IF pressSectionLowerFeltOverrunOperatorSideAlarm THEN
    alarmsDisplay.pressSectionLowerFeltOverrunOperatorSideAlarm := TRUE;
END_IF

IF pressSectionLowerFeltOverrunDriveSideAlarm THEN
    alarmsDisplay.pressSectionLowerFeltOverrunDriveSideAlarm := TRUE;
END_IF


//────────────────────────────────────────────
// PRESS SECTION — GROUP FAULT
//────────────────────────────────────────────
IF pressSectionGroupFaultAlarm THEN
    alarmsDisplay.pressSectionGroupFaultAlarm := TRUE;
END_IF
END_METHOD

METHOD _03_DryingSectionAlarms
VAR_INPUT
END_VAR
(*
    // ─────────────── LUBRIFICATION PUMPS ───────────────
    lubricationPump1FaultAlarm              : BOOL;  // Lubrication pump 1 fault / trip
    lubricationPump2FaultAlarm              : BOOL;  // Lubrication pump 2 fault / trip
    lubricationMinPressureFaultAlarm        : BOOL;  // Minimum pressure not reached / trip
    lubricationMaxPressureFaultAlarm        : BOOL;  // Overpressure in lubrication circuit / trip
	lubricationTankHighTemperatureAlarm 	: BOOL;
	lubricationCircuitHighTemperatureAlarm 	: BOOL;
*)
//==============================================================
// DRYING SECTION — GROUP 1
//==============================================================

//----------------------------
// Drives — Upper (G1)
//----------------------------
IF 	dryingSectionSafetyAlarm THEN
	
	alarmsDisplay.dryingSectionSafetyAlarm := TRUE;
	
END_IF


IF dryingSectionGroup1UpperMasterFaultAlarm THEN
    alarmsDisplay.dryingSectionGroup1UpperMasterFaultAlarm := TRUE;
END_IF

IF dryingSectionGroup1UpperMasterCoolingFaultAlarm THEN
    alarmsDisplay.dryingSectionGroup1UpperMasterCoolingFaultAlarm := TRUE;
END_IF

IF dryingSectionGroup1UpperSlave1FaultAlarm THEN
    alarmsDisplay.dryingSectionGroup1UpperSlave1FaultAlarm := TRUE;
END_IF

IF dryingSectionGroup1UpperSlave1CoolingFaultAlarm THEN
    alarmsDisplay.dryingSectionGroup1UpperSlave1CoolingFaultAlarm := TRUE;
END_IF

IF dryingSectionGroup1UpperSlave2FaultAlarm THEN
    alarmsDisplay.dryingSectionGroup1UpperSlave2FaultAlarm := TRUE;
END_IF

IF dryingSectionGroup1UpperSlave2CoolingFaultAlarm THEN
    alarmsDisplay.dryingSectionGroup1UpperSlave2CoolingFaultAlarm := TRUE;
END_IF

//----------------------------
// Drives — Lower (G1)
//----------------------------
IF dryingSectionGroup1LowerMasterFaultAlarm THEN
    alarmsDisplay.dryingSectionGroup1LowerMasterFaultAlarm := TRUE;
END_IF

IF dryingSectionGroup1LowerMasterCoolingFaultAlarm THEN
    alarmsDisplay.dryingSectionGroup1LowerMasterCoolingFaultAlarm := TRUE;
END_IF

IF dryingSectionGroup1LowerSlave1FaultAlarm THEN
    alarmsDisplay.dryingSectionGroup1LowerSlave1FaultAlarm := TRUE;
END_IF

IF dryingSectionGroup1LowerSlave1CoolingFaultAlarm THEN
    alarmsDisplay.dryingSectionGroup1LowerSlave1CoolingFaultAlarm := TRUE;
END_IF

IF dryingSectionGroup1LowerSlave2FaultAlarm THEN
    alarmsDisplay.dryingSectionGroup1LowerSlave2FaultAlarm := TRUE;
END_IF

IF dryingSectionGroup1LowerSlave2CoolingFaultAlarm THEN
    alarmsDisplay.dryingSectionGroup1LowerSlave2CoolingFaultAlarm := TRUE;
END_IF

//----------------------------
// Fabric overrun protection (G1)
//----------------------------
IF upperDryingSectionGroup1FabricOverrunOperatorSideAlarm THEN
    alarmsDisplay.upperDryingSectionGroup1FabricOverrunOperatorSideAlarm := TRUE;
END_IF

IF upperDryingSectionGroup1FabricOverrunDriveSideAlarm THEN
    alarmsDisplay.upperDryingSectionGroup1FabricOverrunDriveSideAlarm := TRUE;
END_IF

IF lowerDryingSectionGroup1FabricOverrunOperatorSideAlarm THEN
    alarmsDisplay.lowerDryingSectionGroup1FabricOverrunOperatorSideAlarm := TRUE;
END_IF

IF lowerDryingSectionGroup1FabricOverrunDriveSideAlarm THEN
    alarmsDisplay.lowerDryingSectionGroup1FabricOverrunDriveSideAlarm := TRUE;
END_IF

//----------------------------
// Fabric stretcher (G1)
//----------------------------
IF upperDryingSectionGroup1FabricStretcherMotorFaultAlarm THEN
    alarmsDisplay.upperDryingSectionGroup1FabricStretcherMotorFaultAlarm := TRUE;
END_IF

IF lowerDryingSectionGroup1FabricStretcherMotorFaultAlarm THEN
    alarmsDisplay.lowerDryingSectionGroup1FabricStretcherMotorFaultAlarm := TRUE;
END_IF

//----------------------------
// Auxiliaries (G1)
//----------------------------
IF dryingSectionGroup1PickUpRollPosFaultAlarm THEN
    alarmsDisplay.dryingSectionGroup1PickUpRollPosFaultAlarm := TRUE;
END_IF

IF dryingSectionGroup1BabyDryerScraperOscFaultAlarm THEN
    alarmsDisplay.dryingSectionGroup1BabyDryerScraperOscFaultAlarm := TRUE;
END_IF

IF dryingSectionGroup1UpperScraperOscFaultAlarm THEN
    alarmsDisplay.dryingSectionGroup1UpperScraperOscFaultAlarm := TRUE;
END_IF

IF dryingSectionGroup1LowerScraperOscFaultAlarm THEN
    alarmsDisplay.dryingSectionGroup1LowerScraperOscFaultAlarm := TRUE;
END_IF

dryingSectionGroup1PaperBreakAlarm := alarmsDisplay.dryingSectionGroup1PaperBreakAlarm;


//==============================================================
// DRYING SECTION — GROUP 2
//==============================================================

//----------------------------
// Drives — Upper (G2)
//----------------------------
IF dryingSectionGroup2UpperMasterFaultAlarm THEN
    alarmsDisplay.dryingSectionGroup2UpperMasterFaultAlarm := TRUE;
END_IF

IF dryingSectionGroup2UpperMasterCoolingFaultAlarm THEN
    alarmsDisplay.dryingSectionGroup2UpperMasterCoolingFaultAlarm := TRUE;
END_IF

IF dryingSectionGroup2UpperSlave1FaultAlarm THEN
    alarmsDisplay.dryingSectionGroup2UpperSlave1FaultAlarm := TRUE;
END_IF

IF dryingSectionGroup2UpperSlave1CoolingFaultAlarm THEN
    alarmsDisplay.dryingSectionGroup2UpperSlave1CoolingFaultAlarm := TRUE;
END_IF

IF dryingSectionGroup2UpperSlave2FaultAlarm THEN
    alarmsDisplay.dryingSectionGroup2UpperSlave2FaultAlarm := TRUE;
END_IF

IF dryingSectionGroup2UpperSlave2CoolingFaultAlarm THEN
    alarmsDisplay.dryingSectionGroup2UpperSlave2CoolingFaultAlarm := TRUE;
END_IF

//----------------------------
// Drives — Lower (G2)
//----------------------------
IF dryingSectionGroup2LowerMasterFaultAlarm THEN
    alarmsDisplay.dryingSectionGroup2LowerMasterFaultAlarm := TRUE;
END_IF

IF dryingSectionGroup2LowerMasterCoolingFaultAlarm THEN
    alarmsDisplay.dryingSectionGroup2LowerMasterCoolingFaultAlarm := TRUE;
END_IF

IF dryingSectionGroup2LowerSlave1FaultAlarm THEN
    alarmsDisplay.dryingSectionGroup2LowerSlave1FaultAlarm := TRUE;
END_IF

IF dryingSectionGroup2LowerSlave1CoolingFaultAlarm THEN
    alarmsDisplay.dryingSectionGroup2LowerSlave1CoolingFaultAlarm := TRUE;
END_IF

IF dryingSectionGroup2LowerSlave2FaultAlarm THEN
    alarmsDisplay.dryingSectionGroup2LowerSlave2FaultAlarm := TRUE;
END_IF

IF dryingSectionGroup2LowerSlave2CoolingFaultAlarm THEN
    alarmsDisplay.dryingSectionGroup2LowerSlave2CoolingFaultAlarm := TRUE;
END_IF

//----------------------------
// Fabric overrun protection (G2)
//----------------------------
IF upperDryingSectionGroup2FabricOverrunOperatorSideAlarm THEN
    alarmsDisplay.upperDryingSectionGroup2FabricOverrunOperatorSideAlarm := TRUE;
END_IF

IF upperDryingSectionGroup2FabricOverrunDriveSideAlarm THEN
    alarmsDisplay.upperDryingSectionGroup2FabricOverrunDriveSideAlarm := TRUE;
END_IF

IF lowerDryingSectionGroup2FabricOverrunOperatorSideAlarm THEN
    alarmsDisplay.lowerDryingSectionGroup2FabricOverrunOperatorSideAlarm := TRUE;
END_IF

IF lowerDryingSectionGroup2FabricOverrunDriveSideAlarm THEN
    alarmsDisplay.lowerDryingSectionGroup2FabricOverrunDriveSideAlarm := TRUE;
END_IF

//----------------------------
// Fabric stretcher (G2)
//----------------------------
IF upperDryingSectionGroup2FabricStretcherMotorFaultAlarm THEN
    alarmsDisplay.upperDryingSectionGroup2FabricStretcherMotorFaultAlarm := TRUE;
END_IF

IF lowerDryingSectionGroup2FabricStretcherMotorFaultAlarm THEN
    alarmsDisplay.lowerDryingSectionGroup2FabricStretcherMotorFaultAlarm := TRUE;
END_IF

//----------------------------
// Auxiliaries (G2)
//----------------------------
IF dryingSectionGroup2PickUpRollPosFaultAlarm THEN
    alarmsDisplay.dryingSectionGroup2PickUpRollPosFaultAlarm := TRUE;
END_IF

IF dryingSectionGroup2BabyDryerScraperOscFaultAlarm THEN
    alarmsDisplay.dryingSectionGroup2BabyDryerScraperOscFaultAlarm := TRUE;
END_IF

IF dryingSectionGroup2UpperScraperOscFaultAlarm THEN
    alarmsDisplay.dryingSectionGroup2UpperScraperOscFaultAlarm := TRUE;
END_IF

IF dryingSectionGroup2LowerScraperOscFaultAlarm THEN
    alarmsDisplay.dryingSectionGroup2LowerScraperOscFaultAlarm := TRUE;
END_IF

IF dryingSectionGroup2PaperBreakAlarm THEN
    alarmsDisplay.dryingSectionGroup2PaperBreakAlarm := TRUE;
END_IF


//==============================================================
// DRYING SECTION — GROUP 3
//==============================================================

//----------------------------
// Drives — Upper (G3)
//----------------------------
IF dryingSectionGroup3UpperMasterFaultAlarm THEN
    alarmsDisplay.dryingSectionGroup3UpperMasterFaultAlarm := TRUE;
END_IF

IF dryingSectionGroup3UpperMasterCoolingFaultAlarm THEN
    alarmsDisplay.dryingSectionGroup3UpperMasterCoolingFaultAlarm := TRUE;
END_IF

IF dryingSectionGroup3UpperSlave1FaultAlarm THEN
    alarmsDisplay.dryingSectionGroup3UpperSlave1FaultAlarm := TRUE;
END_IF

IF dryingSectionGroup3UpperSlave1CoolingFaultAlarm THEN
    alarmsDisplay.dryingSectionGroup3UpperSlave1CoolingFaultAlarm := TRUE;
END_IF

IF dryingSectionGroup3UpperSlave2FaultAlarm THEN
    alarmsDisplay.dryingSectionGroup3UpperSlave2FaultAlarm := TRUE;
END_IF

IF dryingSectionGroup3UpperSlave2CoolingFaultAlarm THEN
    alarmsDisplay.dryingSectionGroup3UpperSlave2CoolingFaultAlarm := TRUE;
END_IF

//----------------------------
// Drives — Lower (G3)
//----------------------------
IF dryingSectionGroup3LowerMasterFaultAlarm THEN
    alarmsDisplay.dryingSectionGroup3LowerMasterFaultAlarm := TRUE;
END_IF

IF dryingSectionGroup3LowerMasterCoolingFaultAlarm THEN
    alarmsDisplay.dryingSectionGroup3LowerMasterCoolingFaultAlarm := TRUE;
END_IF

IF dryingSectionGroup3LowerSlave1FaultAlarm THEN
    alarmsDisplay.dryingSectionGroup3LowerSlave1FaultAlarm := TRUE;
END_IF

IF dryingSectionGroup3LowerSlave1CoolingFaultAlarm THEN
    alarmsDisplay.dryingSectionGroup3LowerSlave1CoolingFaultAlarm := TRUE;
END_IF

IF dryingSectionGroup3LowerSlave2FaultAlarm THEN
    alarmsDisplay.dryingSectionGroup3LowerSlave2FaultAlarm := TRUE;
END_IF

IF dryingSectionGroup3LowerSlave2CoolingFaultAlarm THEN
    alarmsDisplay.dryingSectionGroup3LowerSlave2CoolingFaultAlarm := TRUE;
END_IF

//----------------------------
// Fabric overrun protection (G3)
//----------------------------
IF upperDryingSectionGroup3FabricOverrunOperatorSideAlarm THEN
    alarmsDisplay.upperDryingSectionGroup3FabricOverrunOperatorSideAlarm := TRUE;
END_IF

IF upperDryingSectionGroup3FabricOverrunDriveSideAlarm THEN
    alarmsDisplay.upperDryingSectionGroup3FabricOverrunDriveSideAlarm := TRUE;
END_IF

IF lowerDryingSectionGroup3FabricOverrunOperatorSideAlarm THEN
    alarmsDisplay.lowerDryingSectionGroup3FabricOverrunOperatorSideAlarm := TRUE;
END_IF

IF lowerDryingSectionGroup3FabricOverrunDriveSideAlarm THEN
    alarmsDisplay.lowerDryingSectionGroup3FabricOverrunDriveSideAlarm := TRUE;
END_IF

//----------------------------
// Fabric stretcher (G3)
//----------------------------
IF upperDryingSectionGroup3FabricStretcherMotorFaultAlarm THEN
    alarmsDisplay.upperDryingSectionGroup3FabricStretcherMotorFaultAlarm := TRUE;
END_IF

IF lowerDryingSectionGroup3FabricStretcherMotorFaultAlarm THEN
    alarmsDisplay.lowerDryingSectionGroup3FabricStretcherMotorFaultAlarm := TRUE;
END_IF

//----------------------------
// Auxiliaries (G3)
//----------------------------
IF dryingSectionGroup3PickUpRollPosFaultAlarm THEN
    alarmsDisplay.dryingSectionGroup3PickUpRollPosFaultAlarm := TRUE;
END_IF

IF dryingSectionGroup3BabyDryerScraperOscFaultAlarm THEN
    alarmsDisplay.dryingSectionGroup3BabyDryerScraperOscFaultAlarm := TRUE;
END_IF

IF dryingSectionGroup3UpperScraperOscFaultAlarm THEN
    alarmsDisplay.dryingSectionGroup3UpperScraperOscFaultAlarm := TRUE;
END_IF

IF dryingSectionGroup3LowerScraperOscFaultAlarm THEN
    alarmsDisplay.dryingSectionGroup3LowerScraperOscFaultAlarm := TRUE;
END_IF

IF dryingSectionGroup3PaperBreakAlarm THEN
    alarmsDisplay.dryingSectionGroup3PaperBreakAlarm := TRUE;
END_IF

IF lubricationMinPressureFaultAlarm THEN
	
	alarmsDisplay.lubricationMinPressureFaultAlarm := TRUE;
	
END_IF

IF lubricationMaxPressureFaultAlarm THEN
	
	alarmsDisplay.lubricationMaxPressureFaultAlarm := TRUE;
	
END_IF



IF lubricationPump1FaultAlarm THEN
	
	alarmsDisplay.lubricationPump1FaultAlarm := TRUE;
	
END_IF

IF lubricationPump2FaultAlarm THEN
	
	alarmsDisplay.lubricationPump2FaultAlarm := TRUE;
	
END_IF

IF lubricationTankHighTemperatureAlarm THEN
	
	alarmsDisplay.lubricationTankHighTemperatureAlarm := TRUE;
	
END_IF


IF lubricationCircuitHighTemperatureAlarm THEN
	
	alarmsDisplay.lubricationCircuitHighTemperatureAlarm := TRUE;
	
END_IF
END_METHOD

METHOD _04_WinderSectionAlarms
VAR_INPUT
END_VAR
(*

    // ─────────────── DRYING SECTION — GROUP 1 ───────────────
    dryingSectionGroup1UpperMasterFaultAlarm         : BOOL;  // G1 Upper Master fault / trip
    dryingSectionGroup1UpperMasterCoolingFaultAlarm  : BOOL;  // G1 Upper Master forced cooling fault
    dryingSectionGroup1UpperSlave1FaultAlarm         : BOOL;  // G1 Upper Slave1 fault / trip
    dryingSectionGroup1UpperSlave1CoolingFaultAlarm  : BOOL;  // G1 Upper Slave1 forced cooling fault
    dryingSectionGroup1UpperSlave2FaultAlarm         : BOOL;  // G1 Upper Slave2 fault / trip
    dryingSectionGroup1UpperSlave2CoolingFaultAlarm  : BOOL;  // G1 Upper Slave2 forced cooling fault

    dryingSectionGroup1LowerMasterFaultAlarm         : BOOL;  // G1 Lower Master fault / trip
    dryingSectionGroup1LowerMasterCoolingFaultAlarm  : BOOL;  // G1 Lower Master forced cooling fault
    dryingSectionGroup1LowerSlave1FaultAlarm         : BOOL;  // G1 Lower Slave1 fault / trip
    dryingSectionGroup1LowerSlave1CoolingFaultAlarm  : BOOL;  // G1 Lower Slave1 forced cooling fault
    dryingSectionGroup1LowerSlave2FaultAlarm         : BOOL;  // G1 Lower Slave2 fault / trip
    dryingSectionGroup1LowerSlave2CoolingFaultAlarm  : BOOL;  // G1 Lower Slave2 forced cooling fault

    // ── FABRIC OVERRUN PROTECTION — GROUP 1 ───────────────────────────────────
    upperDryingSectionGroup1FabricOverrunOperatorSideAlarm : BOOL;  // Fabric overrun detected on operator side (sensor active)
    upperDryingSectionGroup1FabricOverrunDriveSideAlarm    : BOOL;  // Fabric overrun detected on drive side (sensor active)
    lowerDryingSectionGroup1FabricOverrunOperatorSideAlarm : BOOL;  // Fabric overrun detected on operator side (sensor active)
    lowerDryingSectionGroup1FabricOverrunDriveSideAlarm    : BOOL;  // Fabric overrun detected on drive side (sensor active)

    // ───────── DRYING SECTION — FABRIC STRETCHER — GROUP 1 ─────────
    upperDryingSectionGroup1FabricStretcherMotorFaultAlarm : BOOL;  // Upper fabric stretcher motor fault (G1)
    lowerDryingSectionGroup1FabricStretcherMotorFaultAlarm : BOOL;  // Lower fabric stretcher motor fault (G1)

    // ───────── DRYING SECTION — AUXILIARIES — GROUP 1 ─────────
    dryingSectionGroup1PickUpRollPosFaultAlarm       : BOOL;  // EN: G1 pick-up roll positioner fault / PT: Falha do posicionador do rolo pick-up G1
    dryingSectionGroup1BabyDryerScraperOscFaultAlarm : BOOL;  // EN: G1 babydryer scraper oscillator fault / PT: Falha do oscilador da raspa do babydryer G1
    dryingSectionGroup1UpperScraperOscFaultAlarm     : BOOL;  // EN: G1 upper group scraper oscillator fault / PT: Falha do oscilador da raspa do grupo superior G1
    dryingSectionGroup1LowerScraperOscFaultAlarm     : BOOL;  // EN: G1 lower group scraper oscillator fault / PT: Falha do oscilador da raspa do grupo inferior G1
    dryingSectionGroup1PaperBreakAlarm     : BOOL;  // EN: G1 lower group scraper oscillator fault / PT: Falha do oscilador da raspa do grupo inferior G1

    // ─────────────── DRYING SECTION — GROUP 2 ───────────────
    dryingSectionGroup2UpperMasterFaultAlarm         : BOOL;  // G2 Upper Master fault / trip
    dryingSectionGroup2UpperMasterCoolingFaultAlarm  : BOOL;  // G2 Upper Master forced cooling fault
    dryingSectionGroup2UpperSlave1FaultAlarm         : BOOL;  // G2 Upper Slave1 fault / trip
    dryingSectionGroup2UpperSlave1CoolingFaultAlarm  : BOOL;  // G2 Upper Slave1 forced cooling fault
    dryingSectionGroup2UpperSlave2FaultAlarm         : BOOL;  // G2 Upper Slave2 fault / trip
    dryingSectionGroup2UpperSlave2CoolingFaultAlarm  : BOOL;  // G2 Upper Slave2 forced cooling fault

    dryingSectionGroup2LowerMasterFaultAlarm         : BOOL;  // G2 Lower Master fault / trip
    dryingSectionGroup2LowerMasterCoolingFaultAlarm  : BOOL;  // G2 Lower Master forced cooling fault
    dryingSectionGroup2LowerSlave1FaultAlarm         : BOOL;  // G2 Lower Slave1 fault / trip
    dryingSectionGroup2LowerSlave1CoolingFaultAlarm  : BOOL;  // G2 Lower Slave1 forced cooling fault
    dryingSectionGroup2LowerSlave2FaultAlarm         : BOOL;  // G2 Lower Slave2 fault / trip
    dryingSectionGroup2LowerSlave2CoolingFaultAlarm  : BOOL;  // G2 Lower Slave2 forced cooling fault

    // ── FABRIC OVERRUN PROTECTION — GROUP 2 ───────────────────────────────────
    upperDryingSectionGroup2FabricOverrunOperatorSideAlarm : BOOL;  // Fabric overrun detected on operator side (sensor active)
    upperDryingSectionGroup2FabricOverrunDriveSideAlarm    : BOOL;  // Fabric overrun detected on drive side (sensor active)
    lowerDryingSectionGroup2FabricOverrunOperatorSideAlarm : BOOL;  // Fabric overrun detected on operator side (sensor active)
    lowerDryingSectionGroup2FabricOverrunDriveSideAlarm    : BOOL;  // Fabric overrun detected on drive side (sensor active)

    // ───────── DRYING SECTION — FABRIC STRETCHER — GROUP 2 ─────────
    upperDryingSectionGroup2FabricStretcherMotorFaultAlarm : BOOL;  // Upper fabric stretcher motor fault (G2)
    lowerDryingSectionGroup2FabricStretcherMotorFaultAlarm : BOOL;  // Lower fabric stretcher motor fault (G2)

    // ───────── DRYING SECTION — AUXILIARIES — GROUP 2 ─────────
    dryingSectionGroup2PickUpRollPosFaultAlarm       : BOOL;  // EN: G2 pick-up roll positioner fault / PT: Falha do posicionador do rolo pick-up G2
    dryingSectionGroup2BabyDryerScraperOscFaultAlarm : BOOL;  // EN: G2 babydryer scraper oscillator fault / PT: Falha do oscilador da raspa do babydryer G2
    dryingSectionGroup2UpperScraperOscFaultAlarm     : BOOL;  // EN: G2 upper group scraper oscillator fault / PT: Falha do oscilador da raspa do grupo superior G2
    dryingSectionGroup2LowerScraperOscFaultAlarm     : BOOL;  // EN: G2 lower group scraper oscillator fault / PT: Falha do oscilador da raspa do grupo inferior G2
    dryingSectionGroup2PaperBreakAlarm     : BOOL;  // EN: G1 lower group scraper oscillator fault / PT: Falha do oscilador da raspa do grupo inferior G1

    // ─────────────── DRYING SECTION — GROUP 3 ───────────────
    dryingSectionGroup3UpperMasterFaultAlarm         : BOOL;  // G3 Upper Master fault / trip
    dryingSectionGroup3UpperMasterCoolingFaultAlarm  : BOOL;  // G3 Upper Master forced cooling fault
    dryingSectionGroup3UpperSlave1FaultAlarm         : BOOL;  // G3 Upper Slave1 fault / trip
    dryingSectionGroup3UpperSlave1CoolingFaultAlarm  : BOOL;  // G3 Upper Slave1 forced cooling fault
    dryingSectionGroup3UpperSlave2FaultAlarm         : BOOL;  // G3 Upper Slave2 fault / trip
    dryingSectionGroup3UpperSlave2CoolingFaultAlarm  : BOOL;  // G3 Upper Slave2 forced cooling fault

    dryingSectionGroup3LowerMasterFaultAlarm         : BOOL;  // G3 Lower Master fault / trip
    dryingSectionGroup3LowerMasterCoolingFaultAlarm  : BOOL;  // G3 Lower Master forced cooling fault
    dryingSectionGroup3LowerSlave1FaultAlarm         : BOOL;  // G3 Lower Slave1 fault / trip
    dryingSectionGroup3LowerSlave1CoolingFaultAlarm  : BOOL;  // G3 Lower Slave1 forced cooling fault
    dryingSectionGroup3LowerSlave2FaultAlarm         : BOOL;  // G3 Lower Slave2 fault / trip
    dryingSectionGroup3LowerSlave2CoolingFaultAlarm  : BOOL;  // G3 Lower Slave2 forced cooling fault

    // ── FABRIC OVERRUN PROTECTION — GROUP 3 ───────────────────────────────────
    upperDryingSectionGroup3FabricOverrunOperatorSideAlarm : BOOL;  // Fabric overrun detected on operator side (sensor active)
    upperDryingSectionGroup3FabricOverrunDriveSideAlarm    : BOOL;  // Fabric overrun detected on drive side (sensor active)
    lowerDryingSectionGroup3FabricOverrunOperatorSideAlarm : BOOL;  // Fabric overrun detected on operator side (sensor active)
    lowerDryingSectionGroup3FabricOverrunDriveSideAlarm    : BOOL;  // Fabric overrun detected on drive side (sensor active)

    // ───────── DRYING SECTION — FABRIC STRETCHER — GROUP 3 ─────────
    upperDryingSectionGroup3FabricStretcherMotorFaultAlarm : BOOL;  // Upper fabric stretcher motor fault (G3)
    lowerDryingSectionGroup3FabricStretcherMotorFaultAlarm : BOOL;  // Lower fabric stretcher motor fault (G3)

    // ───────── DRYING SECTION — AUXILIARIES — GROUP 3 ─────────
    dryingSectionGroup3PickUpRollPosFaultAlarm       : BOOL;  // EN: G3 pick-up roll positioner fault / PT: Falha do posicionador do rolo pick-up G3
    dryingSectionGroup3BabyDryerScraperOscFaultAlarm : BOOL;  // EN: G3 babydryer scraper oscillator fault / PT: Falha do oscilador da raspa do babydryer G3
    dryingSectionGroup3UpperScraperOscFaultAlarm     : BOOL;  // EN: G3 upper group scraper oscillator fault / PT: Falha do oscilador da raspa do grupo superior G3
    dryingSectionGroup3LowerScraperOscFaultAlarm     : BOOL;  // EN: G3 lower group scraper oscillator fault / PT: Falha do oscilador da raspa do grupo inferior G3
    dryingSectionGroup3PaperBreakAlarm     : BOOL;  // EN: G1 lower group scraper oscillator fault / PT: Falha do oscilador da raspa do grupo inferior G1

*)
//==============================================================
// DRYING SECTION — GROUP 1
//==============================================================

//----------------------------
// Drives — Upper (G1)
//----------------------------
IF 	winderSectionSafetyAlarm THEN
	
	alarmsDisplay.winderSectionSafetyAlarm := TRUE;
	
END_IF
END_METHOD

METHOD _08_AlarmIndication

VAR
	
	alarmCompResult	: DINT;

END_VAR

alarmCompResult := MEMCMP(pBuf1:= ADR(alarmsVariables) , pBuf2:= ADR(alarmsDisplay) , n:= SIZEOF(alarmsDisplay));

//alarmCompResult := alarmsVariables <> alarmsDisplay;

IF alarmCompResult <> 0 THEN

	alarmIndication := TRUE;
ELSE
	
	alarmIndication := FALSE;
	
END_IF
END_METHOD

END_FUNCTION_BLOCK

// ---- Function Blocks/DELTA - MS300/FB_DELTA_C2000_ETC.TcPOU
FUNCTION_BLOCK FB_DELTA_C2000_ETC



//======================================================================
// Persistent Configuration Inputs
//======================================================================
VAR_INPUT PERSISTENT
	
    deviceConfig            : C2000_DEV_CONFIG;       // Device-specific configuration (scaling, limits, etc.)

END_VAR

//======================================================================
// Runtime Inputs
//======================================================================
VAR_INPUT
	
    speedSetpoint           : REAL;                		// Motor speed reference to be written to drive
	torqueSetpoint			: REAL;						// Torque limit if running as torque
    commandWord             : C2000_CONTROLWORD;      	// Control word to drive (start, stop, etc.)
    digitalOutputs          : C2000_DIGITAL_OUTPUTS;  	// Digital output values to send to drive
    analogOutputs           : C2000_ANALOG_OUTPUTS;   	// Analog output values to send to drive
	
END_VAR

//======================================================================
// Runtime Outputs
//======================================================================
VAR_OUTPUT
	
    statusWord              : C2000_STATUSWORD;       // Current status word read from drive
    digitalInputs           : C2000_DIGITAL_INPUTS;   // Current status of digital inputs from drive
    analogInputs            : C2000_ANALOG_INPUTS;    // Current status of analog inputs from drive
    motorSpeedRPM             : REAL;                   // Actual motor speed read from drive in RPM
    motorSpeedEng             : REAL;                   // Actual motor speed read from drive in enginering units scaled
    outputCurrent           : REAL;                   // Output current read from drive
    outputTorque            : REAL;                   // Output torque read from drive
	
	
	pdoSpeedSet			: INT;
	
	
END_VAR

//======================================================================
// Internal Variables
//======================================================================
VAR
    PDOS                    : C2000_PDOS;             // Process Data Object structure containing drive mappings
    // One-shot + pulse for fault reset
    rTrigReset : R_TRIG;
    tReset     : TOF;
	
    // Base OMS bits default (keep your logic)
    b0_swOn, b1_enVolt, b2_qStopOK, b3_enOp : BOOL;
    b4, b5, b6, b7_faultReset, b8_halt      : BOOL;
    cw                                       : WORD;

    // Reset sequencer helpers
 //   rTrigReset        : R_TRIG;   // detect rising edge of reset command
    tResetClear       : TON;      // phase 1: clear all bits (control word = 0)
    tResetPulse       : TON;      // phase 2: pulse bit7 = 1
    resetSeqActive    : BOOL;     // TRUE while running either phase
    resetClearPt      : TIME := T#500MS;    // adjust if your drive needs longer clear
    resetPulsePt      : TIME := T#1000ms;  // 1 second fault-reset pulse	

END_VAR

(*==============================================================================================================================
CPNTeck - Automação Industrial
(c)Copyright 2025 All Rights Reserved
_______________________________________________________________________________________________________________________________
Library: N/A
Tested with: CX920
Engineering: TwinCAT 3
Restrictions: -
Requirements: N/A
Functionality: This function block communicates with a Delta MS300 drive over Modbus RTU. It reads process values such as
               motor speed, current, torque, status words, digital and analog inputs, and writes control commands and 
               setpoints to the drive. The block includes timeout monitoring and state-based communication handling.
Support: fabio@cpnteck.com.br
Note: Parameter comments are only available in language 'English (United States)'

_______________________________________________________________________________________________________________________________
Change log table:

Version         | Date         | Expert in charge   | Changes applied
01.00.01        | 31.05.2025   | Fabio Campion      | Initial implementation for MS300 drive Modbus RTU communication
==============================================================================================================================*)

_StatusWord();       // Method to handle the status word of the drive
_DigitalInputs();    // Method to process the status of digital inputs
_AnalogInputs();     // Method to handle analog input values

_CommandWord();      // Method to set or process the command word for the drive
_DigitalOutputs();   // Method to manage the status of digital outputs
_AnalogOutputs();    // Method to handle analog output values
_SetOperationMode();
_FeedBackVariables(); // Method to process feedback variables from the drive
_SpeedReference();         // Method to set or process the setpoint values
_TorqueReference();

METHOD PRIVATE _AnalogInputs
VAR_INPUT
END_VAR
END_METHOD

METHOD PRIVATE _AnalogOutputs
VAR_INPUT
END_VAR
END_METHOD

METHOD PRIVATE _CommandWord
VAR_INPUT
END_VAR
(*
VAR
    // Internal
    b0_swOn, b1_enVolt, b2_qStopOK, b3_enOp, b4, b5, b6 : BOOL;
    b7_faultReset, b8_halt                              : BOOL;
    cw                                                  : UINT;
END_VAR
*)

b4 := 1;
b5 := 1;
b6 := 1;


// ---------- 1) Base state from commands (bits 0..3) ----------
IF commandWord.quickStop THEN
    // Quick-stop has highest priority: keep voltage/switch-on, clear enable op, force bit2=0
    b0_swOn    := TRUE;
    b1_enVolt  := TRUE;
    b2_qStopOK := FALSE;  // bit2=0 => quick stop active
    b3_enOp    := FALSE;

ELSIF commandWord.enableDrive THEN
    // Enable Operation: 1,1,1,1
    b0_swOn    := TRUE;
    b1_enVolt  := TRUE;
    b2_qStopOK := TRUE;
    b3_enOp    := TRUE;

ELSIF commandWord.stopRequest THEN
    // Switch On (ready but not enabled): 1,1,1,0
    b0_swOn    := TRUE;
    b1_enVolt  := TRUE;
    b2_qStopOK := TRUE;
    b3_enOp    := FALSE;

ELSE
    // Shutdown (safe, DC bus on): 0,1,1,0
    b0_swOn    := FALSE;
    b1_enVolt  := TRUE;
    b2_qStopOK := TRUE;
    b3_enOp    := FALSE;
END_IF


// ---------- 2) Halt (bit8) ----------
b8_halt := commandWord.halt;

// ---------- 3) Fault Reset as 1000 ms pulse (bit7) ----------
rTrigReset(CLK := commandWord.faultResetCmd);
tReset(IN := rTrigReset.Q, PT := T#1000ms);
b7_faultReset := tReset.Q;

// ---------- 4) Pack bits into 16-bit control word ----------
cw := 0; // bits 9..15 remain 0 unless you set them later

// base (0..3)
IF b0_swOn    THEN cw := cw OR 16#0001; END_IF; // bit0
IF b1_enVolt  THEN cw := cw OR 16#0002; END_IF; // bit1
IF b2_qStopOK THEN cw := cw OR 16#0004; END_IF; // bit2
IF b3_enOp    THEN cw := cw OR 16#0008; END_IF; // bit3

// OMS (4..6) — use correct masks
IF b4          THEN cw := cw OR 16#0010; END_IF; // bit4
IF b5          THEN cw := cw OR 16#0020; END_IF; // bit5
IF b6          THEN cw := cw OR 16#0040; END_IF; // bit6

// bit7 (fault reset pulse) and bit8 (halt)
IF b7_faultReset THEN cw := cw OR 16#0080; END_IF; // bit7
IF b8_halt       THEN cw := cw OR 16#0100; END_IF; // bit8

// Bits 9..15 reserved = 0
PDOS.PlcToDrv.controlWord := cw;



//==============================================================
// CIA402 CONTROL WORD BUILD — with proper reset sequence
//==============================================================
(*

//==============================================================
// 0) Edge-detect RESET command and run the two-phase sequence
//==============================================================
rTrigReset(CLK := commandWord.faultResetCmd);

// Start sequence on rising edge
IF rTrigReset.Q THEN
    resetSeqActive := TRUE;
    // (Re)start clear phase
    tResetClear(IN := TRUE, PT := resetClearPt);
    // ensure pulse is off until clear finishes
    tResetPulse(IN := FALSE, PT := resetPulsePt);
END_IF;

// Advance/reset timers when sequence is active
IF resetSeqActive THEN
    // Phase 1: CLEAR (control word = 0)
    tResetClear(IN := tResetClear.IN, PT := resetClearPt);

    // When clear finishes, start pulse (only once)
    IF tResetClear.Q AND NOT tResetPulse.IN THEN
        tResetClear(IN := FALSE, PT := resetClearPt);     // stop clear timer
        tResetPulse(IN := TRUE,  PT := resetPulsePt);     // start pulse
    END_IF;

    // Run pulse
    tResetPulse(IN := tResetPulse.IN, PT := resetPulsePt);

    // Sequence ends when pulse finishes
    IF tResetPulse.Q THEN
        tResetPulse(IN := FALSE, PT := resetPulsePt);
        resetSeqActive := FALSE;
    END_IF;
END_IF;


//==============================================================
// 1) NORMAL PACKING (only used when NOT resetting)
//==============================================================

// Default OMS high (per your original)
b4 := TRUE;  // bit4 mask 0x0010
b5 := TRUE;  // bit5 mask 0x0020
b6 := TRUE;  // bit6 mask 0x0040

// ---------- 1) Base state from commands (bits 0..3) ----------
IF commandWord.quickStop THEN
    // Quick-stop has highest priority
    b0_swOn    := TRUE;
    b1_enVolt  := TRUE;
    b2_qStopOK := FALSE; // quick stop active
    b3_enOp    := FALSE;

ELSIF commandWord.enableDrive THEN
    // Enable Operation: 1,1,1,1
    b0_swOn    := TRUE;
    b1_enVolt  := TRUE;
    b2_qStopOK := TRUE;
    b3_enOp    := TRUE;

ELSIF commandWord.stopRequest THEN
    // Switch On (ready but not enabled): 1,1,1,0
    b0_swOn    := TRUE;
    b1_enVolt  := TRUE;
    b2_qStopOK := TRUE;
    b3_enOp    := FALSE;

ELSE
    // Shutdown (safe, DC bus on): 0,1,1,0
    b0_swOn    := FALSE;
    b1_enVolt  := TRUE;
    b2_qStopOK := TRUE;
    b3_enOp    := FALSE;
END_IF;

// ---------- 2) Halt (bit8) ----------
b8_halt := commandWord.halt;


//==============================================================
// 2) BUILD CONTROL WORD — with RESET SEQUENCE OVERRIDE
//==============================================================
cw := 0;

// If reset sequence is active, override everything
IF resetSeqActive THEN
    // Phase 1: CLEAR → send 0x0000
    IF NOT tResetClear.Q THEN
//        cw := 16#0000;
        cw := 16#0080;
		

    // Phase 2: PULSE → send only bit7 = 1 (0x0080)
    ELSIF tResetClear.Q AND NOT tResetPulse.Q THEN
//        cw := 16#0080;
        cw := 16#0000;
		
    END_IF;

ELSE
    // Normal packing
    // base (0..3)
    IF b0_swOn    THEN cw := cw OR 16#0001; END_IF; // bit0
    IF b1_enVolt  THEN cw := cw OR 16#0002; END_IF; // bit1
    IF b2_qStopOK THEN cw := cw OR 16#0004; END_IF; // bit2
    IF b3_enOp    THEN cw := cw OR 16#0008; END_IF; // bit3

    // OMS (4..6)
    IF b4          THEN cw := cw OR 16#0010; END_IF; // bit4
    IF b5          THEN cw := cw OR 16#0020; END_IF; // bit5
    IF b6          THEN cw := cw OR 16#0040; END_IF; // bit6

    // bit7 (fault reset) — now driven EXCLUSIVELY by the sequencer, so keep low here
    // b7_faultReset := FALSE;

    // bit8 (halt)
    IF b8_halt       THEN cw := cw OR 16#0100; END_IF; // bit8

    // Bits 9..15 remain 0 unless set elsewhere
END_IF;

// Push to PDO
PDOS.PlcToDrv.controlWord := cw;
*)
END_METHOD

METHOD PRIVATE _DigitalInputs 
VAR_INPUT
END_VAR
END_METHOD

METHOD PRIVATE _DigitalOutputs : BOOL
VAR_INPUT
END_VAR
END_METHOD

METHOD PRIVATE _FeedBackVariables
VAR_INPUT
END_VAR

VAR
	
	OutputTorqueAux : REAL;

END_VAR
// Calculate the actual motor speed
motorSpeedRPM := DINT_TO_REAL(PDOS.DrvToPLC.velocityActualValue);
// Calculate the actual motor speed in meters per minute
motorSpeedEng := _Scale(
    X := DINT_TO_REAL(PDOS.DrvToPLC.velocityActualValue), 
    I_LO := deviceConfig.MotorSpeedInputLow, 
    I_HI := deviceConfig.MotorSpeedInputHigh, 
    O_LO := deviceConfig.MotorSpeedMPMOutputLow, 
    O_HI := deviceConfig.MotorSpeedMPMOutputHigh
);

// Calculate the actual output torque
OutputTorque := _Scale(
    X := INT_TO_REAL(PDOS.DrvToPLC.torqueActualValue), 
    I_LO := deviceConfig.OutputTorqueInputLow, 
    I_HI := deviceConfig.OutputTorqueInputHigh, 
    O_LO := deviceConfig.OutputTorqueOutputLow, 
    O_HI := deviceConfig.OutputTorqueOutputHigh
);
END_METHOD

METHOD PRIVATE _Scale : REAL
VAR_INPUT
	
	X : REAL;
	I_LO : REAL;
	I_HI : REAL;
	O_LO : REAL;
	O_HI : REAL;
	
END_VAR
IF I_LO = I_HI THEN
	_Scale := O_LO;
ELSE
	_Scale := (O_HI - O_LO) / (I_HI - I_LO) * (LIMIT(I_LO, X, I_HI) - I_LO) + O_LO;
END_IF;
END_METHOD

METHOD PRIVATE _SetOperationMode
VAR_INPUT
END_VAR
CASE deviceConfig.operationMode OF

    E_C2000_ModeOfOperation.Reserved_0:
        PDOS.PlcToDrv.modesOfOperation := 0;
        ; // Reserved - no action

    E_C2000_ModeOfOperation.ProfilePositionMode:
        PDOS.PlcToDrv.modesOfOperation := 1;
        ; // Profile Position Mode handling

    E_C2000_ModeOfOperation.VelocityMode:
        PDOS.PlcToDrv.modesOfOperation := 2;
        ; // Velocity Mode handling

    E_C2000_ModeOfOperation.Reserved_3:
        PDOS.PlcToDrv.modesOfOperation := 3;
        ; // Reserved - no action

    E_C2000_ModeOfOperation.ProfileTorqueMode:
        PDOS.PlcToDrv.modesOfOperation := 4;
		
        ; // Profile Torque Mode handling

    E_C2000_ModeOfOperation.Reserved_5:
        PDOS.PlcToDrv.modesOfOperation := 5;
        ; // Reserved - no action

    E_C2000_ModeOfOperation.HomingMode:
        PDOS.PlcToDrv.modesOfOperation := 6;
        ; // Homing Mode handling

    E_C2000_ModeOfOperation.Reserved_7:
        PDOS.PlcToDrv.modesOfOperation := 7;
        ; // Reserved - no action

    E_C2000_ModeOfOperation.CyclicSynchronousPositionMode:
        PDOS.PlcToDrv.modesOfOperation := 8;
        ; // Cyclic Synchronous Position Mode handling

    E_C2000_ModeOfOperation.Reserved_9:
        PDOS.PlcToDrv.modesOfOperation := 9;
        ; // Reserved - no action

    E_C2000_ModeOfOperation.CyclicSynchronousTorqueMode:
        PDOS.PlcToDrv.modesOfOperation := 10;
        ; // Cyclic Synchronous Torque Mode handling

ELSE
    PDOS.PlcToDrv.modesOfOperation := 2;
    ; // Fallback: Undefined mode, default to reserved

END_CASE
END_METHOD

METHOD PRIVATE _SpeedReference
VAR_INPUT
END_VAR
// --- Update Velocity Target Setpoint (signed INT) ---
PDOS.PlcToDrv.vlTargetVelocity := REAL_TO_INT(_Scale(
    X    := speedSetpoint, 
    I_LO := deviceConfig.speedSetpointInputLow, 
    I_HI := deviceConfig.speedSetpointInputHigh, 
    O_LO := deviceConfig.speedSetpointOutputLow, 
    O_HI := deviceConfig.speedSetpointOutputHigh));

	PDOS.PlcToDrv.maxMotorSpeed := PDOS.PlcToDrv.vlTargetVelocity;
	
	pdoSpeedSet := PDOS.PlcToDrv.vlTargetVelocity;
END_METHOD

METHOD PRIVATE _StatusWord
VAR_INPUT
END_VAR
// --- Map raw statusword bits to structured fields ---------------------------
StatusWord.readyToSwitchOn     := PDOS.DrvToPLC.StatusWord.0;   // Bit 0
StatusWord.switchedOn          := PDOS.DrvToPLC.StatusWord.1;   // Bit 1
StatusWord.operationEnabled    := PDOS.DrvToPLC.StatusWord.2;   // Bit 2
StatusWord.fault               := PDOS.DrvToPLC.StatusWord.3;   // Bit 3
StatusWord.voltageEnabled      := PDOS.DrvToPLC.StatusWord.4;   // Bit 4
StatusWord.quickStop           := PDOS.DrvToPLC.StatusWord.5;   // Bit 5
StatusWord.switchOnDisabled    := PDOS.DrvToPLC.StatusWord.6;   // Bit 6
StatusWord.warning             := PDOS.DrvToPLC.StatusWord.7;   // Bit 7
StatusWord.reserved1           := PDOS.DrvToPLC.StatusWord.8;   // Bit 8 (reserved)
StatusWord.remote              := PDOS.DrvToPLC.StatusWord.9;   // Bit 9
StatusWord.targetReached       := PDOS.DrvToPLC.StatusWord.10;  // Bit 10
StatusWord.internalLimitActive := PDOS.DrvToPLC.StatusWord.11;  // Bit 11
END_METHOD

METHOD PRIVATE _TorqueReference
VAR_INPUT
END_VAR

VAR
END_VAR


IF deviceConfig.torqueLimiterEnabled THEN
	
	// --- Update Velocity Target Setpoint (signed INT) ---
	PDOS.PlcToDrv.maxTorque := REAL_TO_UINT(_Scale(
		X    := torqueSetpoint, 
		I_LO := deviceConfig.torqueSetpointInputLow, 
		I_HI := deviceConfig.torqueSetpointInputHigh, 
		O_LO := deviceConfig.torqueSetpointOutputLow, 
		O_HI := deviceConfig.torqueSetpointOutputHigh) + deviceConfig.torqueDif);
		
ELSE
	
	PDOS.PlcToDrv.maxTorque := REAL_TO_UINT (deviceConfig.torqueSetpointOutputHigh);
	
END_IF
END_METHOD

END_FUNCTION_BLOCK

// ---- Function Blocks/IOs/Beckhoff/EL1809 - Digital Inputs/FB_EL1809.TcPOU
FUNCTION_BLOCK FB_EL1809
VAR_INPUT

	deviceConfig    : EL1809_DEV_CONFIG; // Configuration settings for the CT121F device
	
END_VAR
VAR_OUTPUT
		
	digitalInput_01  : BOOL;
	digitalInput_02  : BOOL;
	digitalInput_03  : BOOL;
	digitalInput_04  : BOOL;
	digitalInput_05  : BOOL;
	digitalInput_06  : BOOL;
	digitalInput_07  : BOOL;
	digitalInput_08  : BOOL;
	digitalInput_09  : BOOL;
	digitalInput_10  : BOOL;
	digitalInput_11  : BOOL;
	digitalInput_12  : BOOL;
	digitalInput_13  : BOOL;
	digitalInput_14  : BOOL;
	digitalInput_15  : BOOL;
	digitalInput_16  : BOOL;


END_VAR
VAR
	    PDOS : EL1809_HWTOPLC_PDOS; // Process Data Objects for RWPT01D communication
END_VAR


inputState();

METHOD PRIVATE inputState
// Inputs Mapping Configuration

digitalInput_01 		:= PDOS.digitalInput_01 OR (deviceConfig.enableForce AND deviceConfig.forceDigitalInput_00);
digitalInput_02 		:= PDOS.digitalInput_02 OR (deviceConfig.enableForce AND deviceConfig.forceDigitalInput_01);
digitalInput_03 		:= PDOS.digitalInput_03 OR (deviceConfig.enableForce AND deviceConfig.forceDigitalInput_02);
digitalInput_04 		:= PDOS.digitalInput_04 OR (deviceConfig.enableForce AND deviceConfig.forceDigitalInput_03);
digitalInput_05 		:= PDOS.digitalInput_05 OR (deviceConfig.enableForce AND deviceConfig.forceDigitalInput_04);
digitalInput_06 		:= PDOS.digitalInput_06 OR (deviceConfig.enableForce AND deviceConfig.forceDigitalInput_05);
digitalInput_07	 		:= PDOS.digitalInput_07 OR (deviceConfig.enableForce AND deviceConfig.forceDigitalInput_06);
digitalInput_08 		:= PDOS.digitalInput_08 OR (deviceConfig.enableForce AND deviceConfig.forceDigitalInput_07);
digitalInput_09 		:= PDOS.digitalInput_09 OR (deviceConfig.enableForce AND deviceConfig.forceDigitalInput_08);
digitalInput_10 		:= PDOS.digitalInput_10 OR (deviceConfig.enableForce AND deviceConfig.forceDigitalInput_09);
digitalInput_11 		:= PDOS.digitalInput_11 OR (deviceConfig.enableForce AND deviceConfig.forceDigitalInput_10);
digitalInput_12 		:= PDOS.digitalInput_12 OR (deviceConfig.enableForce AND deviceConfig.forceDigitalInput_11);
digitalInput_13 		:= PDOS.digitalInput_13 OR (deviceConfig.enableForce AND deviceConfig.forceDigitalInput_12);
digitalInput_14 		:= PDOS.digitalInput_14 OR (deviceConfig.enableForce AND deviceConfig.forceDigitalInput_13);
digitalInput_15 		:= PDOS.digitalInput_15 OR (deviceConfig.enableForce AND deviceConfig.forceDigitalInput_14);
digitalInput_16 		:= PDOS.digitalInput_16 OR (deviceConfig.enableForce AND deviceConfig.forceDigitalInput_15);
END_METHOD

END_FUNCTION_BLOCK

// ---- Function Blocks/IOs/Beckhoff/EL2809 - Digital Outputs/FB_EL2809.TcPOU
FUNCTION_BLOCK FB_EL2809
VAR_INPUT
	


	deviceConfig    : EL2809_DEV_CONFIG; // Configuration settings for the CT222F device
	
	digitalOutput_01 : BOOL;
	digitalOutput_02 : BOOL;
	digitalOutput_03 : BOOL;
	digitalOutput_04 : BOOL;
	digitalOutput_05 : BOOL;
	digitalOutput_06 : BOOL;
	digitalOutput_07 : BOOL;
	digitalOutput_08 : BOOL;
	digitalOutput_09 : BOOL;
	digitalOutput_10 : BOOL;
	digitalOutput_11 : BOOL;
	digitalOutput_12 : BOOL;
	digitalOutput_13 : BOOL;
	digitalOutput_14 : BOOL;
	digitalOutput_15 : BOOL;
	digitalOutput_16 : BOOL;
	
END_VAR
VAR_OUTPUT


END_VAR
VAR
	    PDOS : EL2809_PDOS; // Process Data Objects for RWPT01D communication
END_VAR


outputState();

METHOD PRIVATE outputState
// Outputs Mapping Configuration


PDOS.PlcToHw.digitalOutput_01 := digitalOutput_01 OR (deviceConfig.enableForce AND deviceConfig.forceDigitalOutput_00);
PDOS.PlcToHw.digitalOutput_02 := digitalOutput_02 OR (deviceConfig.enableForce AND deviceConfig.forceDigitalOutput_01);
PDOS.PlcToHw.digitalOutput_03 := digitalOutput_03 OR (deviceConfig.enableForce AND deviceConfig.forceDigitalOutput_02); 
PDOS.PlcToHw.digitalOutput_04 := digitalOutput_04 OR (deviceConfig.enableForce AND deviceConfig.forceDigitalOutput_03); 
PDOS.PlcToHw.digitalOutput_05 := digitalOutput_05 OR (deviceConfig.enableForce AND deviceConfig.forceDigitalOutput_04); 
PDOS.PlcToHw.digitalOutput_06 := digitalOutput_06 OR (deviceConfig.enableForce AND deviceConfig.forceDigitalOutput_05); 
PDOS.PlcToHw.digitalOutput_07 := digitalOutput_07 OR (deviceConfig.enableForce AND deviceConfig.forceDigitalOutput_06); 
PDOS.PlcToHw.digitalOutput_08 := digitalOutput_08 OR (deviceConfig.enableForce AND deviceConfig.forceDigitalOutput_07); 
PDOS.PlcToHw.digitalOutput_09 := digitalOutput_09 OR (deviceConfig.enableForce AND deviceConfig.forceDigitalOutput_08); 
PDOS.PlcToHw.digitalOutput_10 := digitalOutput_10 OR (deviceConfig.enableForce AND deviceConfig.forceDigitalOutput_09); 
PDOS.PlcToHw.digitalOutput_11 := digitalOutput_11 OR (deviceConfig.enableForce AND deviceConfig.forceDigitalOutput_10); 
PDOS.PlcToHw.digitalOutput_12 := digitalOutput_12 OR (deviceConfig.enableForce AND deviceConfig.forceDigitalOutput_11); 
PDOS.PlcToHw.digitalOutput_13 := digitalOutput_13 OR (deviceConfig.enableForce AND deviceConfig.forceDigitalOutput_12); 
PDOS.PlcToHw.digitalOutput_14 := digitalOutput_14 OR (deviceConfig.enableForce AND deviceConfig.forceDigitalOutput_13); 
PDOS.PlcToHw.digitalOutput_15 := digitalOutput_15 OR (deviceConfig.enableForce AND deviceConfig.forceDigitalOutput_14); 
PDOS.PlcToHw.digitalOutput_16 := digitalOutput_16 OR (deviceConfig.enableForce AND deviceConfig.forceDigitalOutput_15);
END_METHOD

END_FUNCTION_BLOCK

// ---- Function Blocks/IOs/Beckhoff/EL3152 - Ai 2 x 4-20MA - 16bit/FB_EL3152.TcPOU
FUNCTION_BLOCK FB_EL3152
VAR_INPUT PERSISTENT

	deviceConfig    : EL3152_DEV_CONFIG; // Configuration settings for the CT121F device
	
END_VAR
VAR_OUTPUT
		
	Channel1  : REAL;
	Channel2  : REAL;
	
END_VAR
VAR
	    PDOS : EL3052_PDOS; // Process Data Objects for RWPT01D communication
END_VAR


_AnalogInputs();

METHOD PRIVATE _AnalogInputs
VAR_INPUT
END_VAR
// Calculate the actual motor speed
Channel1 := _Scale(
    X := DINT_TO_REAL(PDOS.HwToPLC.Channel1.Value), 
    I_LO := deviceConfig.channel1InputLow, 
    I_HI := deviceConfig.channel1InputHigh, 
    O_LO := deviceConfig.channel1OutputLow, 
    O_HI := deviceConfig.channel1OutputHigh
);

// Calculate the actual motor speed
Channel2 := _Scale(
    X := DINT_TO_REAL(PDOS.HwToPLC.Channel2.Value), 
    I_LO := deviceConfig.channe12InputLow, 
    I_HI := deviceConfig.channe12InputHigh, 
    O_LO := deviceConfig.channe12OutputLow, 
    O_HI := deviceConfig.channe12OutputHigh
);
END_METHOD

METHOD PRIVATE _Scale : REAL
VAR_INPUT
	
	X : REAL;
	I_LO : REAL;
	I_HI : REAL;
	O_LO : REAL;
	O_HI : REAL;
	
END_VAR
IF I_LO = I_HI THEN
	_Scale := O_LO;
ELSE
	_Scale := (O_HI - O_LO) / (I_HI - I_LO) * (LIMIT(I_LO, X, I_HI) - I_LO) + O_LO;
END_IF;
END_METHOD

END_FUNCTION_BLOCK

// ---- Function Blocks/PaperMachine/Auxiliary/FB_LevelControl.TcPOU
(*
  FUNCTION_BLOCK FB_LevelControl
  Purpose:
    - Level control with Auto/Manual output (0..100 %).
    - PID (OSCAT CTRL_PID) with bumpless transfer.
    - Optional PT1 input filter.
    - VFD supervision: ready, fault, run feedback with timeout.
    - Safety supervision: E-Stop/guards/safety chain => immediate stop anywhere.
    - Interlocks (process permissives) => NORMAL STOP ONLY.
    - Minimum level supervision with hysteresis & debounce (stop/hold/restart).
    - deviceState: human-readable state string.

  States:
    0=Idle, 10=Starting, 20=Running, 90=Stopping
*)

FUNCTION_BLOCK FB_LevelControl
VAR_INPUT
    // ===== Sequence commands =====
    startCommand            : BOOL;            // Start command
    stopCommand             : BOOL;            // Stop command

    // ===== Mode =====
    autoMode                : BOOL;            // TRUE=Automatic / FALSE=Manual

    // ===== Process signals (LEVEL) =====
    levelFeedbackEng        : REAL;            // Level feedback (engineering units)
    levelSetpointEng        : REAL;            // Setpoint in engineering units

    // ===== Manual output (direct % to final element) =====
    manualOutputPct         : REAL;            // 0..100% manual output

    // ===== PID parameters (OSCAT CTRL_PID) =====
    kp                      : REAL := 1.0;     // proportional gain
    tn                      : REAL := 8.0;     // integral time [s]
    tv                      : REAL := 0.0;     // derivative time [s]

    // ===== Output limits & offset =====
    outLowLimitPct          : REAL := 0.0;
    outHighLimitPct         : REAL := 100.0;
    outputOffsetPct         : REAL := 0.0;     // added to final output

    // ===== PID housekeeping =====
    resetPID                : BOOL;            // reset integrator

    // ===== Input filter (OSCAT PT1) =====
    enableInputFilter       : BOOL := TRUE;
    inputFilterTime         : TIME := T#500ms;
    inputFilterGainK        : REAL := 1.0;

    // ===== Optional scaling (engineering <-> %) =====
    enableScaling           : BOOL := TRUE;
    lvlLoEng                : REAL := 0.0;
    lvlHiEng                : REAL := 100.0;

    // ===== VFD interface & supervision =====
    vfdReady                : BOOL;            // VFD ready/healthy
    vfdRunFeedback          : BOOL;            // VFD RUN feedback
    vfdFaultFeedback        : BOOL;            // VFD fault feedback
    vfdRunFbTimeout         : TIME := T#5s;    // Timeout to receive RUN FB after start

    // ===== SAFETY (true safety only) =====
    safetyOk                : BOOL := TRUE;    // Safety relay / chain OK
    estopOk                 : BOOL := TRUE;    // E-Stop loop OK
    guardClosedOk           : BOOL := TRUE;    // Doors/guards closed

    // ===== INTERLOCKS (process permissives) — NORMAL STOP ONLY =====
    interlock1              : BOOL := TRUE;
    interlock2              : BOOL := TRUE;
    interlock3              : BOOL := TRUE;
    interlock4              : BOOL := TRUE;
    interlock5              : BOOL := TRUE;
    interlock6              : BOOL := TRUE;

    // ===== Minimum level supervision (process permissive) =====
    minLevelEnable          : BOOL := TRUE;    // Enable low-level stop/hold logic
    minLevelStopEng         : REAL := 10.0;    // Trip threshold (Eng units) => stop & hold
    minLevelRestartEng      : REAL := 12.0;    // Release threshold (Eng units) => auto restart
    minLevelTripTime        : TIME := T#1s;    // Level < StopEng for this long to trip
    minLevelReleaseTime     : TIME := T#1s;    // Level > RestartEng for this long to release
END_VAR

VAR_OUTPUT
    running                 : BOOL;            // TRUE only in RUN (use to release other devices)
    controlOutputPct        : REAL;            // 0..100 %
    pidDiff                 : REAL;            // SET - ACT (post-scaling)
    pidLimited              : BOOL;            // TRUE if saturated
    deviceState             : STRING(80);      // Human-readable state
    vfdStartCmdOut          : BOOL;            // Asserted in Starting/Running (VFD START)
    minLevelHoldActive      : BOOL;            // TRUE while in low-level hold
END_VAR

VAR
    // State
    step                    : INT;             // 0=Idle,10=Starting,20=Running,90=Stopping
    startOld                : BOOL;
    rStart                  : BOOL;

    // Internals
    manualCmd               : REAL;
    yPID                    : REAL;

    // Filtered PV (engineering)
    levelFeedbackEngFilt    : REAL;

    // PV/SP in %
    pvPct                   : REAL;
    spPct                   : REAL;

    // Timers / supervision
    tonRunFbWait            : TON;

    // Minimum level timers/flags
    minLevelBelow           : BOOL;
    minLevelAboveRestart    : BOOL;
    tonMinLevelTrip         : TON;
    tonMinLevelRelease      : TON;

    // Instances
    instPID                 : CTRL_PID;
    instPT1                 : FT_PT1;

    // Safety aggregation
    allSafetyOK             : BOOL;

    // Interlock aggregation (process-only)
    anyInterlockOpen        : BOOL;
END_VAR



// ============================ Edges ============================
rStart := startCommand AND NOT startOld;
startOld := startCommand;


// ============================ Aggregations =====================
allSafetyOK := safetyOk AND estopOk AND guardClosedOk;
anyInterlockOpen := NOT (interlock1 AND interlock2 AND interlock3 AND interlock4 AND interlock5 AND interlock6);

// Default each cycle
vfdStartCmdOut := FALSE;


// ============================ Minimum level supervision ============================
// Compare using current engineering PV (raw). If preferred, swap to levelFeedbackEngFilt.
minLevelBelow        := (levelFeedbackEng <  minLevelStopEng);
minLevelAboveRestart := (levelFeedbackEng >  minLevelRestartEng);

IF minLevelEnable THEN
    // Trip debounce
    tonMinLevelTrip(IN := minLevelBelow, PT := minLevelTripTime);
    // Release debounce
    tonMinLevelRelease(IN := minLevelAboveRestart, PT := minLevelReleaseTime);

    // Latch HOLD on trip, clear on release
    IF tonMinLevelTrip.Q THEN
        minLevelHoldActive := TRUE;
    END_IF;
    IF tonMinLevelRelease.Q THEN
        minLevelHoldActive := FALSE;
    END_IF;
ELSE
    tonMinLevelTrip(IN := FALSE);
    tonMinLevelRelease(IN := FALSE);
    minLevelHoldActive := FALSE;
END_IF;


// ============================ Immediate stop / safety/fault guards ============
IF stopCommand THEN
    controlOutputPct := 0.0;
    running := FALSE;
    deviceState := 'Stopping (Stop command)';
    step := 90;
END_IF;

IF vfdFaultFeedback THEN
    deviceState := 'Fault from VFD';
    step := 90;
END_IF;

IF NOT allSafetyOK THEN
    deviceState := 'Stopping: Safety chain open';
    step := 90;
END_IF;


// ============================ State machine =====================
CASE step OF
    // ------------------------------------------------------------
    0: // Idle
        running := FALSE;
        controlOutputPct := 0.0;
        deviceState := 'Idle';
        vfdStartCmdOut := FALSE;

        // Start request
        IF rStart AND NOT stopCommand THEN
            // Safety must be OK; VFD must be ready; min level must not be holding
            IF NOT allSafetyOK THEN
                deviceState := 'Start blocked: Safety not OK';
                step := 0;
            ELSIF NOT vfdReady THEN
                deviceState := 'Start blocked: VFD not ready';
                step := 0;
            ELSIF minLevelEnable AND minLevelHoldActive THEN
                deviceState := 'Start blocked: Low level hold';
                step := 0;
            ELSE
                deviceState := 'Starting';
                vfdStartCmdOut := TRUE;                   // send START to VFD
                tonRunFbWait(IN := TRUE, PT := vfdRunFbTimeout);
                step := 10;
            END_IF
        END_IF

    // ------------------------------------------------------------
    10: // Starting (await RUN feedback)
        running := FALSE;
        deviceState := 'Starting (await RUN fb)';
        vfdStartCmdOut := TRUE;

        // Safety/fault during start => stop
        IF NOT allSafetyOK THEN
            tonRunFbWait(IN := FALSE);
            deviceState := 'Stopping: Safety chain open';
            vfdStartCmdOut := FALSE;
            step := 90;

        ELSIF vfdFaultFeedback THEN
            tonRunFbWait(IN := FALSE);
            deviceState := 'Fault from VFD';
            vfdStartCmdOut := FALSE;
            step := 90;

        // Interlocks are normal stop only
        ELSIF anyInterlockOpen THEN
            tonRunFbWait(IN := FALSE);
            deviceState := 'Stopping: Interlock open';
            vfdStartCmdOut := FALSE;
            step := 90;

        // Minimum level HOLD => normal stop
        ELSIF minLevelEnable AND minLevelHoldActive THEN
            tonRunFbWait(IN := FALSE);
            deviceState := 'Stopping: Low level hold';
            vfdStartCmdOut := FALSE;
            step := 90;

        // RUN fb arrived
        ELSIF vfdRunFeedback THEN
            tonRunFbWait(IN := FALSE);
            step := 20;

        // Timeout
        ELSIF tonRunFbWait.Q THEN
            tonRunFbWait(IN := FALSE);
            deviceState := 'Start failed: RUN feedback timeout';
            vfdStartCmdOut := FALSE;
            step := 90;
        END_IF

    // ------------------------------------------------------------
    20: // Running (control loop)
        running := TRUE;               // release other devices with this
        deviceState := 'Running';
        vfdStartCmdOut := TRUE;

        // Supervision
        IF NOT allSafetyOK THEN
            deviceState := 'Stopping: Safety chain open';
            vfdStartCmdOut := FALSE;
            step := 90;

        ELSIF vfdFaultFeedback THEN
            deviceState := 'Fault from VFD';
            vfdStartCmdOut := FALSE;
            step := 90;

        ELSIF NOT vfdReady THEN
            deviceState := 'Stopping: VFD not ready';
            vfdStartCmdOut := FALSE;
            step := 90;

        ELSIF NOT vfdRunFeedback THEN
            deviceState := 'Stopping: RUN feedback lost';
            vfdStartCmdOut := FALSE;
            step := 90;

        // INTERLOCKS → NORMAL STOP ONLY
        ELSIF anyInterlockOpen THEN
            deviceState := 'Stopping: Interlock open';
            vfdStartCmdOut := FALSE;
            step := 90;

        // Minimum level HOLD → NORMAL STOP
        ELSIF minLevelEnable AND minLevelHoldActive THEN
            deviceState := 'Stopping: Low level hold';
            vfdStartCmdOut := FALSE;
            step := 90;

        ELSIF stopCommand THEN
            deviceState := 'Stopping (Stop command)';
            vfdStartCmdOut := FALSE;
            step := 90;

        ELSE
            // ---- Input filtering (PT1) ----
            IF enableInputFilter THEN
                instPT1(in := levelFeedbackEng, T := inputFilterTime, K := inputFilterGainK, out => levelFeedbackEngFilt);
            ELSE
                levelFeedbackEngFilt := levelFeedbackEng;
            END_IF

            // ---- Engineering -> % scaling ----
            IF enableScaling THEN
                pvPct := _ScaleToPct(levelFeedbackEngFilt, lvlLoEng, lvlHiEng);
                spPct := _ScaleToPct(levelSetpointEng,     lvlLoEng, lvlHiEng);
            ELSE
                pvPct := levelFeedbackEngFilt;    // already %
                spPct := levelSetpointEng;        // already %
            END_IF

            // ---- Manual path and PID with bumpless transfer ----
            manualCmd := LIMIT(0.0, manualOutputPct, 100.0);

            instPID(
                ACT := pvPct,
                SET := spPct,
                M_I := manualCmd,
                MAN := NOT autoMode,
                RST := resetPID,
                KP  := kp,
                TN  := tn,
                TV  := tv,
                LL  := outLowLimitPct,
                LH  := outHighLimitPct,
                Y   => yPID,
                DIFF=> pidDiff,
                LIM => pidLimited
            );

            // Mode select, offset, clamp
            IF autoMode THEN
                controlOutputPct := yPID;
            ELSE
                controlOutputPct := manualCmd;
            END_IF
            controlOutputPct := LIMIT(outLowLimitPct, controlOutputPct + outputOffsetPct, outHighLimitPct);
        END_IF

    // ------------------------------------------------------------
    90: // Stopping (normal, de-energize)
        running := FALSE;
        controlOutputPct := 0.0;
        vfdStartCmdOut := FALSE;
        tonRunFbWait(IN := FALSE);

        // Return to Idle once stop released and safety OK
        IF NOT stopCommand AND allSafetyOK THEN
            deviceState := 'Idle';
            step := 0;
        END_IF

    // ------------------------------------------------------------
    ELSE
        running := FALSE;
        controlOutputPct := 0.0;
        deviceState := 'Idle';
        vfdStartCmdOut := FALSE;
        step := 0;
END_CASE

// ============================ Helper ============================
METHOD PRIVATE _ScaleToPct : REAL
VAR_INPUT
    xEng  : REAL;  // value in engineering units
    loEng : REAL;  // min eng
    hiEng : REAL;  // max eng
END_VAR
VAR
    span : REAL;
    pct  : REAL;
END_VAR

span := hiEng - loEng;
IF span = 0.0 THEN
    _ScaleToPct := 0.0; // avoid div by zero
ELSE
    pct := (xEng - loEng) / span * 100.0;
    _ScaleToPct := LIMIT(0.0, pct, 100.0);
END_IF
END_METHOD

END_FUNCTION_BLOCK

// ---- Function Blocks/PaperMachine/Auxiliary/FB_PaperMachine.TcPOU
FUNCTION_BLOCK FB_PaperMachine
VAR_INPUT
	
	safetyCircuit		: BOOL;
	
END_VAR
VAR_OUTPUT
END_VAR
VAR
END_VAR


VAR_IN_OUT

	formingBoardSuctionRollDrive	: FB_DELTA_C2000_ETC;	
	formingBoardTractionRollDrive	: FB_DELTA_C2000_ETC;	

	stockPumpDrive	: FB_DELTA_C2000_ETC;	
	mixPumpDrive	: FB_DELTA_C2000_ETC;	
	wirePitPumpDrive	: FB_DELTA_C2000_ETC;	
	couchPitPumpDrive	: FB_DELTA_C2000_ETC;	

END_VAR

END_FUNCTION_BLOCK

// ---- Function Blocks/PaperMachine/Auxiliary/FB_SimpleMotorStart.TcPOU
FUNCTION_BLOCK FB_SimpleMotorStart
VAR_INPUT
    // Commands & interlocks
    startCommand                : BOOL;   // Start command (Comando de partida)
    stopCommand                 : BOOL;   // Stop command (Comando de parada)
    sofstarterOK                : BOOL;   // Softstarter healthy/ready (Softstarter ok/pronto)
	fault						: BOOL;
	
    interlock1                  : BOOL;   // External interlock 1 (Intertravamento 1)
    interlock2                  : BOOL;   // External interlock 2 (Intertravamento 2)
    interlock3                  : BOOL;   // External interlock 3 (Intertravamento 3)
    interlock4                  : BOOL;   // External interlock 4 (Intertravamento 4)

    // Feedbacks
    softstarterContactorFb      : BOOL;   // FB - softstarter contactor (Retorno do contator do softstarter)
    lineContactorFb             : BOOL;   // FB - line/bypass contactor (Retorno do contator de linha/bypass)

    // Timers
    startDelayTime              : TIME;   // Ramp-up time before switching to line (Tempo de rampa antes do bypass)
    overlapDelayTime            : TIME;   // Both contactors ON overlap (Sobreposição segura de contatores)
    ssContactorTimeout          : TIME;   // Timeout to get SS contactor FB (Tempo máx. retorno contator softstarter)
    lineContactorTimeout        : TIME;   // Timeout to get Line contactor FB (Tempo máx. retorno contator de linha)

    // Motor current proof
    motorCurrentFeedback        : REAL;   // Measured motor current (Corrente medida do motor)
    minCurrentThreshold         : REAL;   // Minimum current to prove energized (Mínimo para provar energização)
    currentProofTime            : TIME;   // Time current must stay above threshold (Tempo de comprovação)
END_VAR

VAR_OUTPUT
	
    faultActive                 : BOOL;   // Latched fault (Falha latched)
    startSequenceRunning        : BOOL;   // Sequence running (Sequência em execução)
    startSequenceFinished       : BOOL;   // Sequence finished successfully (Sequência concluída)

    softstarterContactor        : BOOL;   // CMD softstarter contactor (Comando contator softstarter)
    lineContactor               : BOOL;   // CMD line/bypass contactor (Comando contator linha/bypass)
    softstarterStart            : BOOL;   // CMD start to softstarter (Comando de start do softstarter)

    deviceState                 : STRING(80); // Human-readable state (Estado textual para diagnóstico)
END_VAR

VAR
    // State & edges
    step                        : INT;    // State machine step (Etapa)
    startCommandOld             : BOOL;
    rStart                      : BOOL;

    // Timers
    tonStartDelay               : TON;    // Ramp-up timer (Rampa)
    tonOverlapDelay             : TON;    // Overlap timer (Sobreposição)
    tonCurrentProof             : TON;    // Current proof timer (Prova de corrente)

    tonSSFbTimeout              : TON;    // Timeout for SS contactor FB
    tonLineFbTimeout            : TON;    // Timeout for Line contactor FB

    // Helpers
    allInterlocksOK             : BOOL;
END_VAR


// ============================ Edges, interlocks, defaults ============================
rStart := startCommand AND NOT startCommandOld;
startCommandOld := startCommand;

allInterlocksOK := interlock1 AND interlock2 AND interlock3 AND interlock4;

// Clear "finished" when a new start is requested or stop asserted
IF rStart OR stopCommand THEN
    startSequenceFinished := FALSE;
END_IF

// Default deviceState (will be overwritten below)
deviceState := 'Idle (Parado)';

// =============================== Fault reset =======================================
// Clear fault when no start request and stop is not held
IF NOT startCommand AND NOT stopCommand THEN
    faultActive := FALSE;
END_IF

// Stop command: immediate safe de-energize (Parada segura imediata)
IF stopCommand THEN
    softstarterStart      := FALSE;
    lineContactor         := FALSE;
    softstarterContactor  := FALSE;

    tonStartDelay(IN:=FALSE);
    tonOverlapDelay(IN:=FALSE);
    tonCurrentProof(IN:=FALSE);
    tonSSFbTimeout(IN:=FALSE);
    tonLineFbTimeout(IN:=FALSE);

    startSequenceRunning  := FALSE;
    step := 0;
END_IF

// ============================= Interlocks & health checks ===========================
// Interlocks must be OK and softstarter OK while sequence
IF startCommand AND NOT allInterlocksOK THEN
    faultActive := TRUE;
    deviceState := 'Fault: interlock open (Falha: intertrav. aberto)';
END_IF

IF startCommand AND NOT sofstarterOK THEN
    faultActive := TRUE;
    deviceState := 'Fault: softstarter not OK (Falha: softstarter NOK)';
END_IF

// If fault is active, do not run sequence
IF faultActive THEN
    softstarterStart      := FALSE;
    lineContactor         := FALSE;
    softstarterContactor  := FALSE;

    tonStartDelay(IN:=FALSE);
    tonOverlapDelay(IN:=FALSE);
    tonCurrentProof(IN:=FALSE);
    tonSSFbTimeout(IN:=FALSE);
    tonLineFbTimeout(IN:=FALSE);

    startSequenceRunning  := FALSE;
    step := 0;
END_IF


// ================================= State machine ===================================
IF startCommand AND NOT faultActive AND sofstarterOK AND allInterlocksOK AND NOT stopCommand THEN
    startSequenceRunning := TRUE;

    CASE step OF
        0: // Idle -> energize softstarter contactor
            deviceState := 'Energizing SS contactor (Acionando contator SS)';
            softstarterContactor := TRUE;

            // timers reset
            tonStartDelay(IN:=FALSE);
            tonOverlapDelay(IN:=FALSE);
            tonCurrentProof(IN:=FALSE);

            // start SS feedback timeout while command is ON and FB is OFF
            tonSSFbTimeout(IN:=NOT softstarterContactorFb, PT:=ssContactorTimeout);

            step := 10;

        10: // Wait SS contactor feedback
            deviceState := 'Waiting SS contactor FB (Aguardando retorno SS)';
            // keep timeout running if still no feedback
            tonSSFbTimeout(IN:=NOT softstarterContactorFb);

            // Timeout fault
            IF tonSSFbTimeout.Q THEN
                faultActive := TRUE;
                deviceState := 'Fault: SS FB timeout (Falha: tempo retorno SS)';
                // force safe
                softstarterStart     := FALSE;
                softstarterContactor := FALSE;
                lineContactor        := FALSE;
                step := 0;
            ELSIF softstarterContactorFb THEN
                softstarterStart := TRUE;                           // Start softstarter
                tonStartDelay(IN:=TRUE, PT:=startDelayTime);        // Start ramp timer
                tonSSFbTimeout(IN:=FALSE);                          // Stop SS timeout
                step := 20;
            END_IF

        20: // Prove motor current while ramping
            deviceState := 'Proving current & ramp (Prova de corrente e rampa)';

            // Current proof: only while current >= threshold
            IF ABS(motorCurrentFeedback) >= minCurrentThreshold THEN
                tonCurrentProof(IN:=TRUE, PT:=currentProofTime);
            ELSE
                tonCurrentProof(IN:=FALSE);
            END_IF

            // Keep ramp timer active
            tonStartDelay(IN:=TRUE);

            // Proceed only when BOTH complete
            IF tonCurrentProof.Q AND tonStartDelay.Q THEN
                deviceState := 'Energizing line contactor (Acionando contator linha)';
                lineContactor := TRUE;

                // start line feedback timeout while command is ON and FB is OFF
                tonLineFbTimeout(IN:=NOT lineContactorFb, PT:=lineContactorTimeout);

                tonCurrentProof(IN:=FALSE); // no longer needed
                step := 30;
            END_IF

        30: // Wait line contactor feedback
            deviceState := 'Waiting line contactor FB (Aguardando retorno linha)';
            // keep timeout running if still no feedback
            tonLineFbTimeout(IN:=NOT lineContactorFb);

            // Timeout fault
            IF tonLineFbTimeout.Q THEN
                faultActive := TRUE;
                deviceState := 'Fault: Line FB timeout (Falha: tempo retorno linha)';
                // safe de-energize SS side and line
                softstarterStart     := FALSE;
                softstarterContactor := FALSE;
                lineContactor        := FALSE;
                step := 0;

            ELSIF lineContactorFb THEN
                deviceState := 'Overlap both contactors (Sobreposição contatores)';
                tonOverlapDelay(IN:=TRUE, PT:=overlapDelayTime); // brief overlap
                tonLineFbTimeout(IN:=FALSE);                     // stop timeout
                step := 40;
            END_IF

        40: // Overlap timing
            deviceState := 'Overlapping... (Sobrepondo...)';
            tonOverlapDelay(IN:=TRUE);
            IF tonOverlapDelay.Q THEN
                softstarterStart     := FALSE;   // Stop softstarter
                softstarterContactor := FALSE;   // Release SS contactor
                tonOverlapDelay(IN:=FALSE);
                deviceState := 'Running on line (Operando em linha)';
                step := 50;
            END_IF

        50: // Running on line
            deviceState := 'Running on line (Operando em linha)';
            startSequenceFinished := TRUE;

            // Stay while start is held; release line on stop
            IF NOT startCommand THEN
                lineContactor := FALSE;
                startSequenceRunning := FALSE;
                deviceState := 'Idle (Parado)';
                step := 0;
            END_IF

        ELSE
            deviceState := 'Idle (Parado)';
            step := 0;
    END_CASE

ELSE
    // No start request / inhibited: ensure safe idle
    startSequenceRunning := FALSE;

    // Keep line latched only if we are in step 50 and startCommand is still ON
    IF step <> 50 THEN
        lineContactor := FALSE;
    END_IF

    // Softstarter side always de-energized when idle
    softstarterStart     := FALSE;
    softstarterContactor := FALSE;

    tonStartDelay(IN:=FALSE);
    tonOverlapDelay(IN:=FALSE);
    tonCurrentProof(IN:=FALSE);
    tonSSFbTimeout(IN:=FALSE);
    tonLineFbTimeout(IN:=FALSE);

    IF NOT startCommand THEN
        deviceState := 'Idle (Parado)';
        step := 0;
    END_IF
END_IF

// ============================================================================
// METHOD: _InputFilter
// OSCAT PT1 filter for PV, with enable/disable and bumpless behavior.
// When disabled, the filter tracks input quickly (tiny T) to avoid bumps.
// ============================================================================
METHOD PRIVATE _InputFilter
VAR_INPUT
    enableFilter   : BOOL;  // TRUE=apply PT1, FALSE=bypass
    rawValue       : REAL;  // Input value to be filtered
    filterTime     : TIME;  // PT1 time constant
    filterGainK    : REAL;  // PT1 gain, typically 1.0
END_VAR
VAR_OUTPUT
    filteredValue  : REAL;  // Filtered (or bypassed) value
END_VAR
VAR
    kUse           : REAL;
    tUse           : TIME;
    yPT1           : REAL;
END_VAR


IF enableFilter THEN
    kUse := filterGainK;
    tUse := filterTime;
ELSE
    // Track input closely for bumpless re-enable
    kUse := 1.0;
    tUse := T#10ms;
END_IF;

instsFT_PT1TInputFilter(
    in  := rawValue,
    T   := tUse,
    K   := kUse,
    out => yPT1
);

// Output selection
IF enableFilter THEN
    filteredValue := yPT1;
ELSE
    filteredValue := rawValue;
END_IF;
END_METHOD

END_FUNCTION_BLOCK

// ---- Function Blocks/PaperMachine/Auxiliary/FB_SpeedDroopControl.TcPOU
FUNCTION_BLOCK FB_SpeedDroopControl
VAR_INPUT

	bManualSpeedCommand : BOOL; (*This comand acts manual speed in the output*)
	fMasterReferenceRPM : REAL;
	fMasterMinRPM : REAL;
	fMasterMaxRPM : REAL;
	fMasterMinMPM  : REAL;
	fMasterMaxMPM  : REAL;
	fSlaveFeedbackRPM : REAL;
	fSlaveMinRPM : REAL;
	fSlaveMaxRPM : REAL;
	fSlaveMinMPM  : REAL;
	fSlaveMaxMPM  : REAL;
	fSlaveGearRatio : REAL;
	fSlaveManSpeedMPM  : REAL;
	fSlaveSpeedDifPct: REAL;

END_VAR

VAR_OUTPUT
(*Slave setpoint variables*)
	fSlaveSetpointRPM  : REAL;	(*Speed reference to the drive*)
	fSlaveSetpointPct  : REAL;	(*Speed reference to the drive*)
(*Slave feedback variables*)

	fSlaveFeedbackMPM  : REAL;
	fSlaveFeedbackPct  : REAL;

	fMasterFeedbackMPM  : REAL;	(*Display speed feedback in PCT*)

	fMasterFeedbackPCT  : REAL;	(*Display speed feedback in PCT*)

END_VAR

VAR
END_VAR

VAR_TEMP
	fSlaveSyncSpeedRPM: REAL;
	fSlaveManSpeedRPM : REAL;
END_VAR

(*Calculate the master reference in MPM*)
(*fMasterFeedbackMPM :=LIMIT(-fMasterMinMPM, F_SCALE_R(fMasterReferenceRPM, fMasterMinRPM,fMasterMaxRPM,fMasterMinMPM, fMasterMaxMPM), fMasterMaxMPM);*)
fMasterFeedbackMPM :=_Scale(fMasterReferenceRPM, fMasterMinRPM,fMasterMaxRPM,fMasterMinMPM, fMasterMaxMPM);


(*Calculate the master reference in percentage*)
fMasterFeedbackPct :=LIMIT(0.0, _Scale(fMasterReferenceRPM, fMasterMinRPM,fMasterMaxRPM,0.0, 100.0), 100.0);

(*Calculate slave speed setpoint in percentage*)
fSlaveSetpointPct := (fMasterFeedbackPCT +  (fMasterFeedbackPCT * (fSlaveSpeedDifPct * 0.01))) * fSlaveGearRatio;

(*Calculate slave speed in meters per minute*)
fSlaveFeedbackMPM :=	_Scale(fSlaveFeedbackRPM, fSlaveMinRPM ,fSlaveMaxRPM, fSlaveMinMPM , fSlaveMaxMPM );

(*Calculate slave output speed in percentage*)
fSlaveFeedbackPCT :=	_Scale(fSlaveFeedbackRPM, fSlaveMinRPM ,fSlaveMaxRPM,0  ,100  );

(*Calculate speed setpoint in sync mode*)
fSlaveSyncSpeedRPM := _Scale(fSlaveSetpointPCT,0.0,100.0,fSlaveMinRPM,fSlaveMaxRPM);

(*Calculate speed setpoint in manual mode*)
fSlaveManSpeedRPM := _Scale(fSlaveManSpeedMPM,fSlaveMinMPM,fSlaveMaxMPM,fSlaveMinRPM,fSlaveMaxRPM);



(*
IF #Start THEN
(* assure range of inputs*)
    #Speed_In_Pct := MAX(IN1 := 0.0, IN2 := #Speed_In_Pct);
ELSE
    #Speed_In_Pct := 0.0;
END_IF;

(*Realiza calculo da velocidade [Velocidade de entrada (0-100%)+Offset de velocidade * 
Fator de realação mecanica*)
(*#Speed_Out_Pct := (#Speed_In_Pct + (#Speed_In_Pct * (#Speed_Out_Offset_Pct * 0.01)))*#Factor;*)
 
 
(*Mostra velocidade em RPM*)
IF #Speed_In_Pct_Max = #Speed_In_Pct_Min THEN
    #Speed_Out_RPM := #Speed_Out_RPM_Min;
    
ELSE
    #Speed_Out_RPM := (#Speed_Out_RPM_Max - #Speed_Out_RPM_Min) / ((#Speed_In_Pct_Max) - (#Speed_In_Pct_Min))
    * LIMIT(MN := (#Speed_In_Pct_Min),IN := (#Speed_Out_Pct), MX := (#Speed_In_Pct_Max));
END_IF;


(*Controle do incremento do passe +/-25%
SU - Slow UP
SD - Slow Down*)
#FB220_TUNE2(SU:= #Offset_Plus,
             SD:= #Offset_Minus,
             Y=>#Speed_Out_Offset_Pct);
(*
#FB217_SRAMP(X:=#Speed_Out_Pct,
             A_UP:= 1.0,
             A_DN := -1.0,
             LIMIT_HIGH:=1000.0,
             LIMIT_LOW:=0.0,
             Y=>#Speed_Out_Pct_RMP); *)


#FB218_RAMP_GEN(SetPoint:=#Speed_Out_Pct,
                Out=>#Speed_Out_Pct_RMP);

*)

METHOD PRIVATE _Scale : REAL
VAR_INPUT
	
	X : REAL;
	I_LO : REAL;
	I_HI : REAL;
	O_LO : REAL;
	O_HI : REAL;
	
END_VAR
IF I_LO = I_HI THEN
	_Scale := O_LO;
ELSE
	_Scale := (O_HI - O_LO) / (I_HI - I_LO) * (LIMIT(I_LO, X, I_HI) - I_LO) + O_LO;
END_IF;
END_METHOD

END_FUNCTION_BLOCK

// ---- Function Blocks/PaperMachine/DriveControl/FB_PressSectionDriveControl_V2_bak.TcPOU
FUNCTION_BLOCK FB_PressSectionDriveControl_V2_bak

VAR_INPUT

    //────────────────────────────────────────────
    // GROUP / INTERLOCKS
    //────────────────────────────────────────────
    startGroup              : BOOL; // Start command (pulse) / Comando de partida (pulso)
    stopGroup               : BOOL; // Stop command (level) / Comando de parada (nível)
    groupReset              : BOOL; // Fault reset / Reset de falhas do grupo
	
    //────────────────────────────────────────────
    // AUXILIARY MOTORS — INDICATORS & COMMANDS
    //────────────────────────────────────────────
    grouSpeedDifIncCmd         : BOOL; // Lamp: offset increasing / Lâmpada: aumento de offset
    grouSpeedDifDecCmd         : BOOL; // Lamp: offset decreasing / Lâmpada: redução de offset
	
    //────────────────────────────────────────────
    // SPEED ADJUSTMENTS / OFFSET TUNING
    //────────────────────────────────────────────
    groupRecoverSpeedCmd    : BOOL; // Recover speed while TRUE / Recuperar velocidade enquanto TRUE


    //────────────────────────────────────────────
    // DRIVE STATUS INPUTS — PRESS SECTION (2 MOTORS)
    //────────────────────────────────────────────
    firstPressReady         : BOOL; // First press (MASTER) ready / Prensa 1 (mestre) pronto
    secondPressReady        : BOOL; // Second press (SLAVE) ready / Prensa 2 (escravo) pronto

    //────────────────────────────────────────────
    // SPEED SETPOINTS / MODE
    //────────────────────────────────────────────
    groupAutoSpeedMPM       : REAL; // Auto mode speed [m/min] / Velocidade em modo automático [m/min]
    groupManualSpeedMPM     : REAL := 50.0; // Manual mode speed / Velocidade em modo manual
    groupSpeedAutoMan       : BOOL; // Speed mode: 0=Manual, 1=Auto / Modo de velocidade: 0=Manual, 1=Automático

    //────────────────────────────────────────────
    // SPEED & TORQUE FEEDBACKS
    //────────────────────────────────────────────
    firstPressSpeedFeedback : REAL; // First press speed feedback / Velocidade medida da prensa 1
    firstPressTorqueFeedback: REAL; // First press torque feedback / Torque da prensa 1
    secondPressSpeedFeedback: REAL; // Second press speed feedback / Velocidade medida da prensa 2
    secondPressTorqueFeedback: REAL; // Second press torque feedback / Torque da prensa 2


    //──── Upper Felt 1 Stretcher ────
    upperFelt1StretcherCmdFwd     : BOOL; // Run forward / Comando para frente
    upperFelt1StretcherCmdRev     : BOOL; // Run reverse / Comando para trás
    upperFelt1StretcherFault      : BOOL; // Fault detected / Falha detectada
    upperFelt1StretcherLimitFwd   : BOOL; // End limit forward / Fim de curso frente
    upperFelt1StretcherLimitRev   : BOOL; // End limit reverse / Fim de curso trás

    //──── Upper Felt 2 Stretcher ────
    upperFelt2StretcherCmdFwd     : BOOL; // Run forward / Comando para frente
    upperFeltt2tretcherCmdRev     : BOOL; // Run reverse / Comando para trás (corrigir nome!)
    upperFeltS2tretcherFault      : BOOL; // Fault detected / Falha detectada
    upperFeltS2tretcherLimitFwd   : BOOL; // End limit forward / Fim de curso frente
    upperFeltS2tretcherLimitRev   : BOOL; // End limit reverse / Fim de curso trás

    //──── Lower Felt Stretcher ────
    lowerFeltStretcherCmdFwd      : BOOL;
    lowerFeltStretcherCmdRev      : BOOL;
    lowerFeltStretcherFault       : BOOL;
    lowerFeltStretcherLimitFwd    : BOOL;
    lowerFeltStretcherLimitRev    : BOOL;

    //──── Upper Infeed Roll ────
    upperInfeedRollCmdFwd         : BOOL;
    upperInfeedRollCmdRev         : BOOL;
    upperInfeedRollFault          : BOOL;
    upperInfeedRollLimitFwd       : BOOL;
    upperInfeedRollLimitRev       : BOOL;

    //──── Lower Infeed Roll ────
    lowerInfeedRollCmdFwd         : BOOL;
    lowerInfeedRollCmdRev         : BOOL;
    lowerInfeedRollFault          : BOOL;
    lowerInfeedRollLimitFwd       : BOOL;
    lowerInfeedRollLimitRev       : BOOL;

    //────────────────────────────────────────────
    // FELT EDGE / RUNNING SAFETY SENSORS
    //────────────────────────────────────────────
    pressSectionUpperFelt1OverrunSensorOperatorSide : BOOL; // Operator side / Lado operador
    pressSectionUpperFelt1OverrunSensorDriveSide    : BOOL; // Drive side / Lado comando

    pressSectionUpperFelt2OverrunSensorOperatorSide : BOOL;
    pressSectionUpperFelt2OverrunSensorDriveSide    : BOOL;

    pressSectionLowerFeltOverrunSensorOperatorSide  : BOOL;
    pressSectionLowerFeltOverrunSensorDriveSide     : BOOL;

	
	machineConfig			:  PaperMachine_TypeHmiConfig;
	
END_VAR



VAR_OUTPUT

    //────────────────────────────────────────────
    // STATE / DIAGNOSTICS
    //────────────────────────────────────────────
    deviceState                 : STRING; // Current state string / Estado atual em texto
    statusCode                  : INT;    // 0=Idle, 1=Starting, 2=Running, 3=Fault
    groupFault                  : BOOL;   // TRUE if any group fault active / Falha geral do grupo


    //────────────────────────────────────────────
    // SPEED REFERENCES (TO DRIVES) AND DISPLAY
    //────────────────────────────────────────────
    firstPressSpeedSetpointRPM  		: REAL; // Master speed reference [%] / Referência de velocidade mestre
    secondPressSpeedSetpointRPM 		: REAL; // Slave speed reference [%] / Referência de velocidade escravo 
	
	firstPressSpeedFeedbackRPM  		: REAL; // Master speed reference [%] / Referência de velocidade mestre
    secondPressSpeedFeedbackRPM 		: REAL; // Slave speed reference [%] / Referência de velocidade escravo 
	
	firstPressSpeedFeedbackMPM  		: REAL; // Master speed reference [%] / Referência de velocidade mestre
    secondPressSpeedFeedbackMPM 		: REAL; // Slave speed reference [%] / Referência de velocidade escravo 

	firstPressTorqueFeedbackPct  		: REAL; // Master speed reference [%] / Referência de velocidade mestre
    secondPressTorqueFeedbackPct 		: REAL; // Slave speed reference [%] / Referência de velocidade escravo 
	
	
	nextGroupSpeedRefMPM        : REAL; // Next group speed [m/min] / Velocidade do próximo grupo [m/min]

    //────────────────────────────────────────────
    // TORQUE REFERENCES / LIMITS (SLAVE)
    //────────────────────────────────────────────
    firstPressTorqueRefPct : REAL; // Torque setpoint for slave / Referência de torque escravo

    //────────────────────────────────────────────
    // DRIVE COMMANDS (ENABLE / RESET)
    //────────────────────────────────────────────
    firstPressDriveEnable        : BOOL; // Enable master drive / Habilita drive mestre
    firstPressDriveReset         : BOOL; // Reset master drive fault / Reset falha drive mestre
    secondPressDriveEnable       : BOOL; // Enable slave drive / Habilita drive escravo
    secondPressDriveReset        : BOOL; // Reset slave drive fault / Reset falha drive escravo

    //────────────────────────────────────────────
    // STATUS CODES (PER DRIVE)
    //────────────────────────────────────────────
    firstPressStatusCode        : INT; // 0=Idle, 1=Start, 2=Run, 3=Fault / Código de status da prensa 1
    secondPressStatusCode       : INT; // Código de status da prensa 2

    //────────────────────────────────────────────
    // AUXILIARY MOTORS — DIRECT START OUTPUTS
    //────────────────────────────────────────────
    upperFelt1StretcherRunFwd   : BOOL; // Run forward / Rodar para frente
    upperFelt1StretcherRunRev   : BOOL; // Run reverse / Rodar para trás

    upperFelt2StretcherRunFwd   : BOOL;
    upperFelt2StretcherRunRev   : BOOL;

    lowerFeltStretcherRunFwd    : BOOL;
    lowerFeltStretcherRunRev    : BOOL;

    upperInfeedRollRunFwd       : BOOL;
    upperInfeedRollRunRev       : BOOL;

    lowerInfeedRollRunFwd       : BOOL;
    lowerInfeedRollRunRev       : BOOL;

    //────────────────────────────────────────────
    // HMI ALARMS STRUCTURE
    //────────────────────────────────────────────
    hmiAlarms                   : PaperMachine_TypeHmiAlarms; // Alarm structure / Estrutura de alarmes

END_VAR




VAR
 
	instFB_GroupDriveControl_V1 : FB_GroupDriveControl_V1;
	instFB_GroupSpeedControl_V1 : FB_GroupSpeedControl_V1;
	instFB_GroupDisplayFilters_V1 : FB_GroupDisplayFilters_V1;
	instFB_GroupTorqueTrimControl_V1 : FB_GroupTorqueTrimControl_V1;

	instFB_GroupTorqueTrimControl_V2: FB_GroupTorqueTrimControl_V2;
	speedDif: REAL;
	speedDifError: BOOL;
END_VAR

VAR PERSISTENT

END_VAR

// ─────────────────────────────────────────────────────────────────────────────
// MAIN CALL SEQUENCE
// ─────────────────────────────────────────────────────────────────────────────

_GroupControl();          // 1) State machine: edges, enables, stop modes
_StateDisplay();
_SpeedDifferenceCheck();  // 4) Speed difference monitor & trip
_auxiliaryControls();

_alarmsDisplay();

METHOD _alarmsDisplay
VAR_INPUT
END_VAR
(*
//==============================================================
// FAULT EVALUATION — PER CONDITION (flags only; no global set)
//==============================================================

//----------------------------
// PRESS SECTION DRIVES
//----------------------------
hmiAlarms.pressSectionFirstPressFaultAlarm  := firstPressVfdFaultFeedback;
hmiAlarms.pressSectionSecondPressFaultAlarm := secondPressVfdFaultFeedback;

//----------------------------
// PRESS SECTION AUXILIARIES
//----------------------------
hmiAlarms.pressSectionUpperFeltStretcherFaultAlarm := upperFelt1StretcherFault;
hmiAlarms.pressSectionLowerFeltStretcherFaultAlarm := lowerFeltStretcherFault;
hmiAlarms.pressSectionUpperInfeedRollFaultAlarm    := upperInfeedRollFault;
hmiAlarms.pressSectionLowerInfeedRollFaultAlarm    := lowerInfeedRollFault;


//==============================================================
// PRESS SECTION — FELT EDGE OVERRUN ALARMS (DIRECT SENSORS)
//==============================================================

hmiAlarms.pressSectionUpperFelt1OverrunOperatorSideAlarm := pressSectionUpperFelt1OverrunSensorOperatorSide;
hmiAlarms.pressSectionUpperFelt1OverrunDriveSideAlarm    := pressSectionUpperFelt1OverrunSensorDriveSide;

hmiAlarms.pressSectionUpperFelt2OverrunOperatorSideAlarm := pressSectionUpperFelt2OverrunSensorOperatorSide;
hmiAlarms.pressSectionUpperFelt2OverrunDriveSideAlarm    := pressSectionUpperFelt2OverrunSensorDriveSide;

hmiAlarms.pressSectionLowerFeltOverrunOperatorSideAlarm := pressSectionLowerFeltOverrunSensorOperatorSide;
hmiAlarms.pressSectionLowerFeltOverrunDriveSideAlarm    := pressSectionLowerFeltOverrunSensorDriveSide;


//----------------------------
// PRESS SECTION GROUP FAULT STATUS
//----------------------------
groupFault :=
    hmiAlarms.pressSectionFirstPressFaultAlarm 
	OR hmiAlarms.pressSectionSecondPressFaultAlarm 
	OR hmiAlarms.pressFelt1OverrunOperatorSideAlarm
	OR hmiAlarms.pressFelt1OverrunDriveSideAlarm
	OR hmiAlarms.pressFelt2OverrunOperatorSideAlarm
	OR hmiAlarms.pressFelt2OverrunDriveSideAlarm
	OR hmiAlarms.pressFelt3OverrunOperatorSideAlarm
	OR hmiAlarms.pressFelt3OverrunDriveSideAlarm;


*)
//==============================================================
// FAULT EVALUATION — PER CONDITION (flags only; no global set)
//==============================================================

//----------------------------
// PRESS SECTION DRIVES
//----------------------------
//hmiAlarms.pressSectionFirstPressFaultAlarm  := firstPressVfdFaultFeedback;
//hmiAlarms.pressSectionSecondPressFaultAlarm := secondPressVfdFaultFeedback;

//----------------------------
// PRESS SECTION AUXILIARIES
//----------------------------
hmiAlarms.pressSectionUpperFeltStretcherFaultAlarm := upperFelt1StretcherFault;
hmiAlarms.pressSectionLowerFeltStretcherFaultAlarm := lowerFeltStretcherFault;
hmiAlarms.pressSectionUpperInfeedRollFaultAlarm    := upperInfeedRollFault;
hmiAlarms.pressSectionLowerInfeedRollFaultAlarm    := lowerInfeedRollFault;


//==============================================================
// PRESS SECTION — FELT EDGE OVERRUN ALARMS (DIRECT SENSORS)
//==============================================================

hmiAlarms.pressSectionUpperFelt1OverrunOperatorSideAlarm := pressSectionUpperFelt1OverrunSensorOperatorSide;
hmiAlarms.pressSectionUpperFelt1OverrunDriveSideAlarm    := pressSectionUpperFelt1OverrunSensorDriveSide;

hmiAlarms.pressSectionUpperFelt2OverrunOperatorSideAlarm := pressSectionUpperFelt2OverrunSensorOperatorSide;
hmiAlarms.pressSectionUpperFelt2OverrunDriveSideAlarm    := pressSectionUpperFelt2OverrunSensorDriveSide;

hmiAlarms.pressSectionLowerFeltOverrunOperatorSideAlarm := pressSectionLowerFeltOverrunSensorOperatorSide;
hmiAlarms.pressSectionLowerFeltOverrunDriveSideAlarm    := pressSectionLowerFeltOverrunSensorDriveSide;


//----------------------------
// PRESS SECTION GROUP FAULT STATUS
//----------------------------
groupFault := hmiAlarms.pressSectionFirstPressFaultAlarm OR
		hmiAlarms.pressSectionSecondPressFaultAlarm OR
		hmiAlarms.pressSectionUpperFelt1OverrunOperatorSideAlarm OR
		hmiAlarms.pressSectionUpperFelt1OverrunDriveSideAlarm OR
		hmiAlarms.pressSectionUpperFelt2OverrunOperatorSideAlarm OR
		hmiAlarms.pressSectionUpperFelt2OverrunDriveSideAlarm OR
		hmiAlarms.pressSectionLowerFeltOverrunOperatorSideAlarm OR
		hmiAlarms.pressSectionLowerFeltOverrunDriveSideAlarm;
END_METHOD

METHOD _auxiliaryControls
VAR_INPUT
END_VAR
//============================
// LOWER FELT STRETCHER
//============================
IF NOT lowerFeltStretcherFault THEN
    IF lowerFeltStretcherCmdFwd AND NOT lowerFeltStretcherCmdRev AND NOT lowerFeltStretcherLimitFwd THEN
        lowerFeltStretcherRunFwd := TRUE;
    ELSE
        lowerFeltStretcherRunFwd := FALSE;
    END_IF;

    IF lowerFeltStretcherCmdRev AND NOT lowerFeltStretcherCmdFwd AND NOT lowerFeltStretcherLimitRev THEN
        lowerFeltStretcherRunRev := TRUE;
    ELSE
        lowerFeltStretcherRunRev := FALSE;
    END_IF;
ELSE
    lowerFeltStretcherRunFwd := FALSE;
    lowerFeltStretcherRunRev := FALSE;
END_IF;


//============================
// UPPER INFEED ROLL
//============================
IF NOT upperInfeedRollFault THEN
    IF upperInfeedRollCmdFwd AND NOT upperInfeedRollCmdRev AND NOT upperInfeedRollLimitFwd THEN
        upperInfeedRollRunFwd := TRUE;
    ELSE
        upperInfeedRollRunFwd := FALSE;
    END_IF;

    IF upperInfeedRollCmdRev AND NOT upperInfeedRollCmdFwd AND NOT upperInfeedRollLimitRev THEN
        upperInfeedRollRunRev := TRUE;
    ELSE
        upperInfeedRollRunRev := FALSE;
    END_IF;
ELSE
    upperInfeedRollRunFwd := FALSE;
    upperInfeedRollRunRev := FALSE;
END_IF;


//============================
// LOWER INFEED ROLL
//============================
IF NOT lowerInfeedRollFault THEN
    IF lowerInfeedRollCmdFwd AND NOT lowerInfeedRollCmdRev AND NOT lowerInfeedRollLimitFwd THEN
        lowerInfeedRollRunFwd := TRUE;
    ELSE
        lowerInfeedRollRunFwd := FALSE;
    END_IF;

    IF lowerInfeedRollCmdRev AND NOT lowerInfeedRollCmdFwd AND NOT lowerInfeedRollLimitRev THEN
        lowerInfeedRollRunRev := TRUE;
    ELSE
        lowerInfeedRollRunRev := FALSE;
    END_IF;
ELSE
    lowerInfeedRollRunFwd := FALSE;
    lowerInfeedRollRunRev := FALSE;
END_IF;


//============================
// UPPER FELT 1 STRETCHER
//============================
IF NOT upperFelt1StretcherFault THEN
    IF upperFelt1StretcherCmdFwd AND NOT upperFelt1StretcherCmdRev AND NOT upperFelt1StretcherLimitFwd THEN
        upperFelt1StretcherRunFwd := TRUE;
    ELSE
        upperFelt1StretcherRunFwd := FALSE;
    END_IF;

    IF upperFelt1StretcherCmdRev AND NOT upperFelt1StretcherCmdFwd AND NOT upperFelt1StretcherLimitRev THEN
        upperFelt1StretcherRunRev := TRUE;
    ELSE
        upperFelt1StretcherRunRev := FALSE;
    END_IF;
ELSE
    upperFelt1StretcherRunFwd := FALSE;
    upperFelt1StretcherRunRev := FALSE;
END_IF;

//============================
// UPPER FELT 2 STRETCHER
//============================
IF NOT upperFeltS2tretcherFault THEN
    IF upperFelt2StretcherCmdFwd AND NOT upperFeltt2tretcherCmdRev AND NOT upperFeltS2tretcherLimitFwd THEN
        upperFelt2StretcherRunFwd := TRUE;
    ELSE
        upperFelt2StretcherRunFwd := FALSE;
    END_IF;

    IF upperFeltt2tretcherCmdRev AND NOT upperFelt2StretcherCmdFwd AND NOT upperFeltS2tretcherLimitRev THEN
        upperFelt2StretcherRunRev := TRUE;
    ELSE
        upperFelt2StretcherRunRev := FALSE;
    END_IF;
ELSE
    upperFelt2StretcherRunFwd := FALSE;
    upperFelt2StretcherRunRev := FALSE;
END_IF;
END_METHOD

METHOD _GroupControl
VAR_INPUT
END_VAR
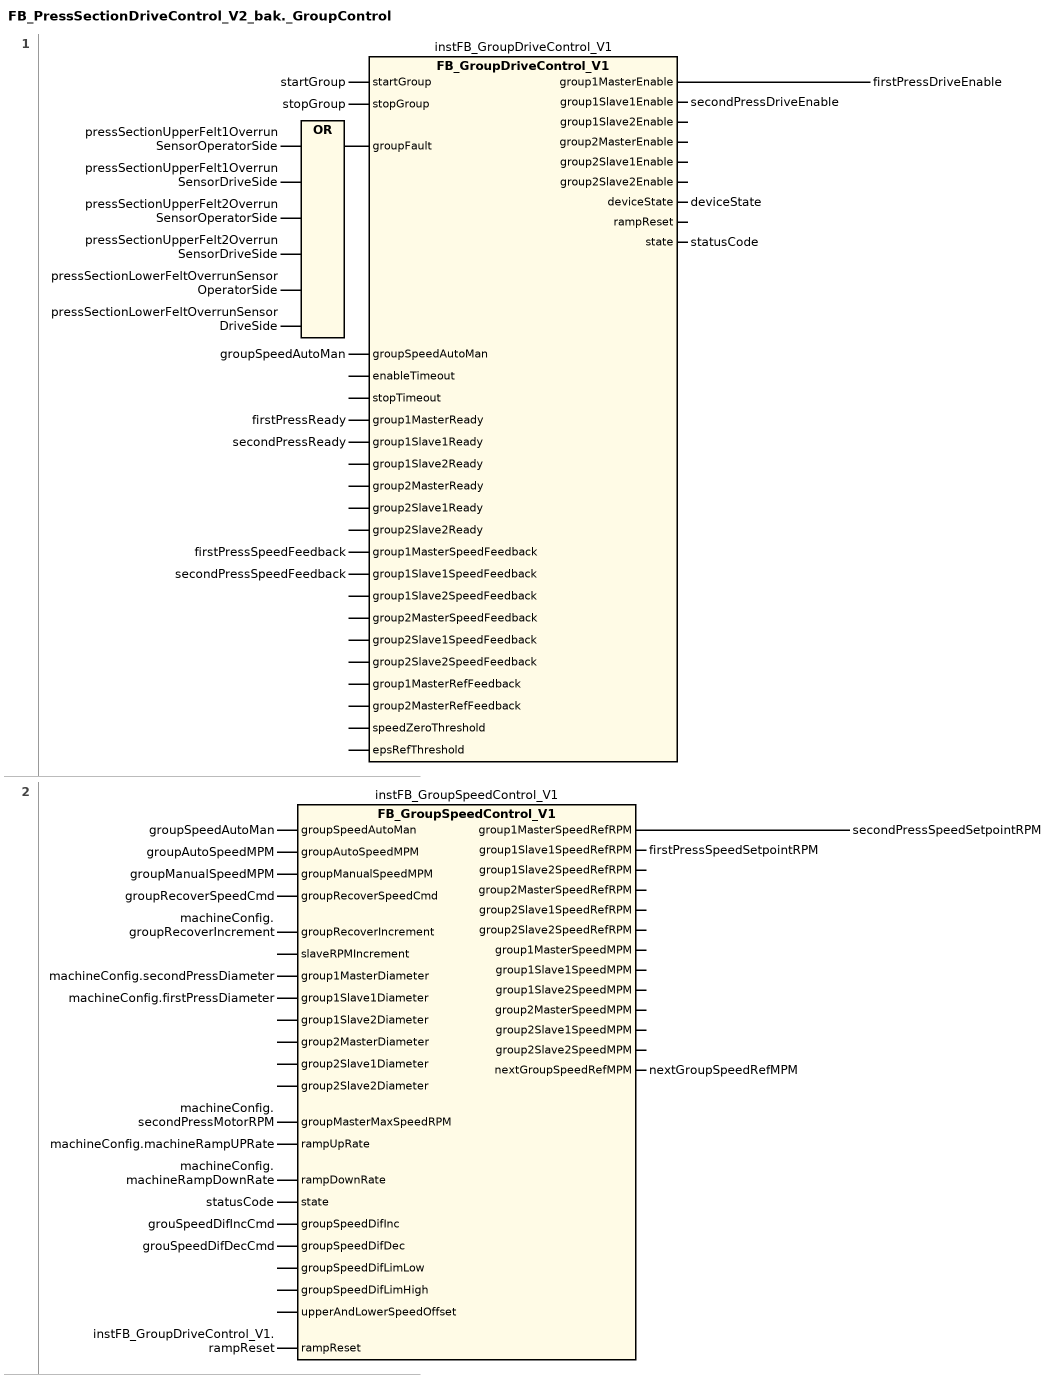
// NETWORK 1
instFB_GroupDriveControl_V1(
    startGroup := startGroup,
    stopGroup := stopGroup,
    groupFault := pressSectionUpperFelt1OverrunSensorOperatorSide OR pressSectionUpperFelt1OverrunSensorDriveSide OR pressSectionUpperFelt2OverrunSensorOperatorSide OR pressSectionUpperFelt2OverrunSensorDriveSide OR pressSectionLowerFeltOverrunSensorOperatorSide OR pressSectionLowerFeltOverrunSensorDriveSide,
    groupSpeedAutoMan := groupSpeedAutoMan,
    group1MasterReady := firstPressReady,
    group1Slave1Ready := secondPressReady,
    group1MasterSpeedFeedback := firstPressSpeedFeedback,
    group1Slave1SpeedFeedback := secondPressSpeedFeedback,
    group1Slave1Enable => secondPressDriveEnable,
    deviceState => deviceState,
    state => statusCode); // FB_GroupDriveControl_V1
firstPressDriveEnable := instFB_GroupDriveControl_V1.group1MasterEnable;

// NETWORK 2
instFB_GroupSpeedControl_V1(
    groupSpeedAutoMan := groupSpeedAutoMan,
    groupAutoSpeedMPM := groupAutoSpeedMPM,
    groupManualSpeedMPM := groupManualSpeedMPM,
    groupRecoverSpeedCmd := groupRecoverSpeedCmd,
    groupRecoverIncrement := machineConfig.groupRecoverIncrement,
    group1MasterDiameter := machineConfig.secondPressDiameter,
    group1Slave1Diameter := machineConfig.firstPressDiameter,
    groupMasterMaxSpeedRPM := machineConfig.secondPressMotorRPM,
    rampUpRate := machineConfig.machineRampUPRate,
    rampDownRate := machineConfig.machineRampDownRate,
    state := statusCode,
    groupSpeedDifInc := grouSpeedDifIncCmd,
    groupSpeedDifDec := grouSpeedDifDecCmd,
    rampReset := instFB_GroupDriveControl_V1.rampReset,
    group1Slave1SpeedRefRPM => firstPressSpeedSetpointRPM,
    nextGroupSpeedRefMPM => nextGroupSpeedRefMPM); // FB_GroupSpeedControl_V1
secondPressSpeedSetpointRPM := instFB_GroupSpeedControl_V1.group1MasterSpeedRefRPM;

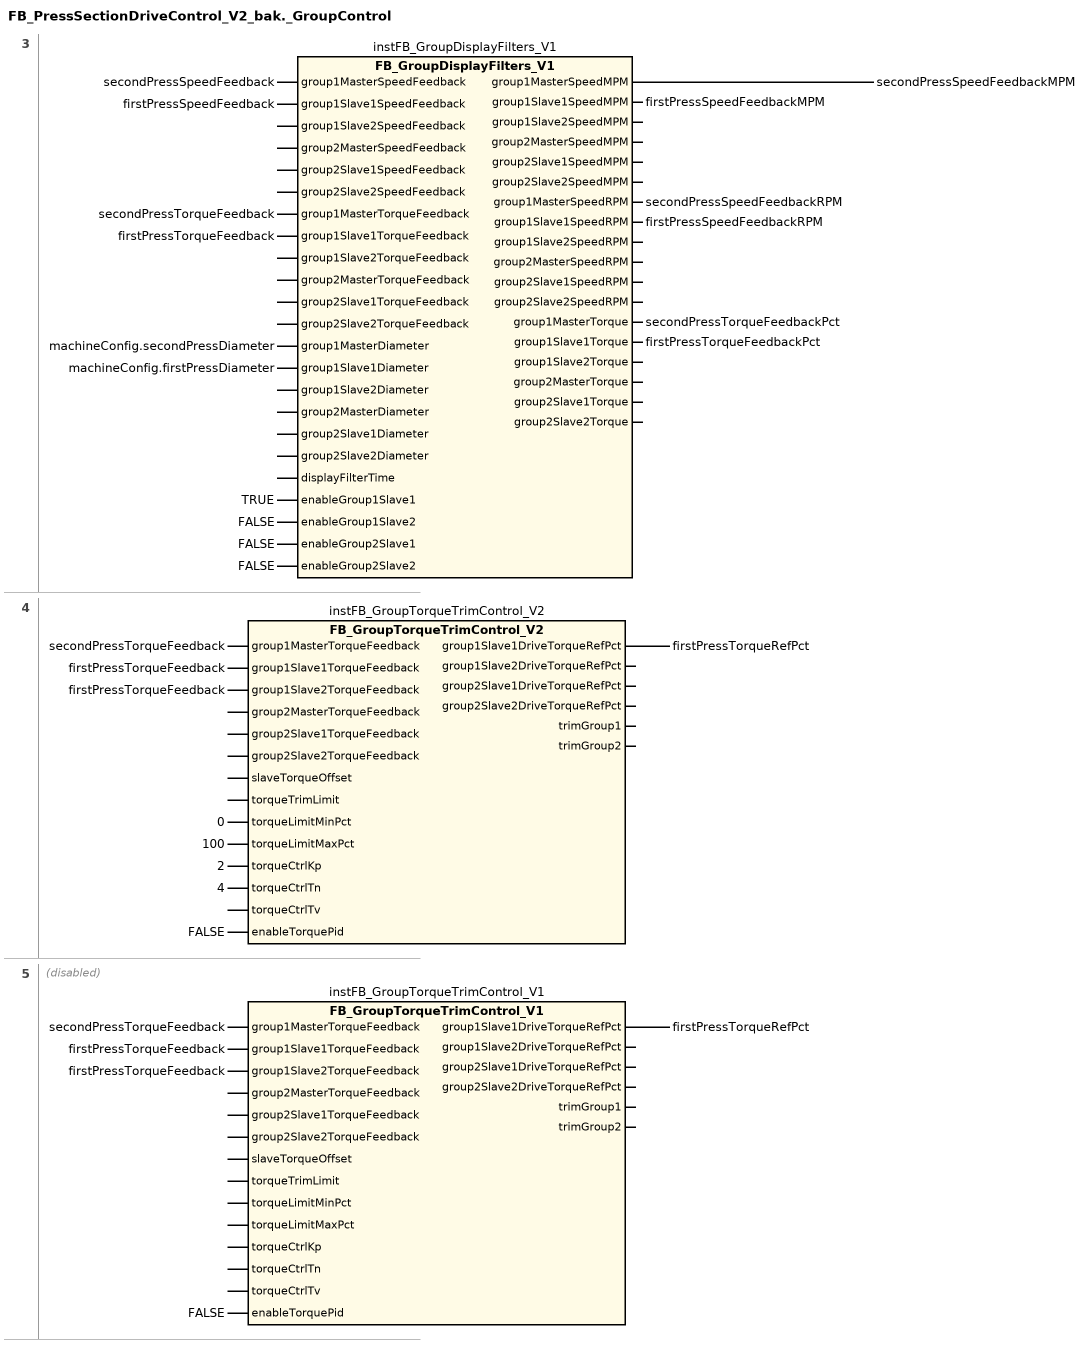
// NETWORK 3
instFB_GroupDisplayFilters_V1(
    group1MasterSpeedFeedback := secondPressSpeedFeedback,
    group1Slave1SpeedFeedback := firstPressSpeedFeedback,
    group1MasterTorqueFeedback := secondPressTorqueFeedback,
    group1Slave1TorqueFeedback := firstPressTorqueFeedback,
    group1MasterDiameter := machineConfig.secondPressDiameter,
    group1Slave1Diameter := machineConfig.firstPressDiameter,
    enableGroup1Slave1 := TRUE,
    enableGroup1Slave2 := FALSE,
    enableGroup2Slave1 := FALSE,
    enableGroup2Slave2 := FALSE,
    group1Slave1SpeedMPM => firstPressSpeedFeedbackMPM,
    group1MasterSpeedRPM => secondPressSpeedFeedbackRPM,
    group1Slave1SpeedRPM => firstPressSpeedFeedbackRPM,
    group1MasterTorque => secondPressTorqueFeedbackPct,
    group1Slave1Torque => firstPressTorqueFeedbackPct); // FB_GroupDisplayFilters_V1
secondPressSpeedFeedbackMPM := instFB_GroupDisplayFilters_V1.group1MasterSpeedMPM;

// NETWORK 4
instFB_GroupTorqueTrimControl_V2(
    group1MasterTorqueFeedback := secondPressTorqueFeedback,
    group1Slave1TorqueFeedback := firstPressTorqueFeedback,
    group1Slave2TorqueFeedback := firstPressTorqueFeedback,
    torqueLimitMinPct := 0,
    torqueLimitMaxPct := 100,
    torqueCtrlKp := 2,
    torqueCtrlTn := 4,
    enableTorquePid := FALSE); // FB_GroupTorqueTrimControl_V2
firstPressTorqueRefPct := instFB_GroupTorqueTrimControl_V2.group1Slave1DriveTorqueRefPct;

// NETWORK 5 (disabled)
// instFB_GroupTorqueTrimControl_V1(
//     group1MasterTorqueFeedback := secondPressTorqueFeedback,
//     group1Slave1TorqueFeedback := firstPressTorqueFeedback,
//     group1Slave2TorqueFeedback := firstPressTorqueFeedback,
//     enableTorquePid := FALSE); // FB_GroupTorqueTrimControl_V1
// firstPressTorqueRefPct := instFB_GroupTorqueTrimControl_V1.group1Slave1DriveTorqueRefPct;
END_METHOD

METHOD PRIVATE _Scale : REAL
VAR_INPUT
    X    : REAL;
    I_LO : REAL;
    I_HI : REAL;
    O_LO : REAL;
    O_HI : REAL;
END_VAR
IF I_LO = I_HI THEN
	_Scale := O_LO;
ELSE
	_Scale := (O_HI - O_LO) / (I_HI - I_LO) * (LIMIT(I_LO, X, I_HI) - I_LO) + O_LO;
END_IF;
END_METHOD

// ============================== Methods ==============================
// Intra-section speed supervision for Press Section (firstPress ↔ secondPress)
METHOD _SpeedDifferenceCheck
VAR_INPUT
END_VAR
VAR
    diffPress : REAL;   // Absolute speed difference between master and slave
END_VAR

(*
    //────────────────────────────────────────────
    firstPressSpeedFeedback : REAL; // First press speed feedback / Velocidade medida da prensa 1
    firstPressTorqueFeedback: REAL; // First press torque feedback / Torque da prensa 1
    secondPressSpeedFeedback: REAL; // Second press speed feedback / Velocidade medida da prensa 2
    secondPressTorqueFeedback: REAL; // Second press torque feedback / Torque da prensa 2

*)


speedDif := ABS(firstPressSpeedFeedback - secondPressSpeedFeedback);


IF speedDif > 10 THEN
	
	speedDifError := TRUE;
	
	ELSE
		
	speedDifError := FALSE;
	
	
END_IF
END_METHOD

METHOD _StateDisplay
VAR_INPUT
END_VAR

// ──────────────────────────────────────────────────────────────────────────────
// _StateDisplay — Press Section (firstPress = Master, secondPress = Slave)
// Maps the internal machine "state" to a compact HMI status code and derives
// per-drive motor status codes from VFD signals.
//
// statusCode / firstPressStatusCode / secondPressStatusCode legend:
//   0 = Idle, 1 = Starting, 2 = Running, 3 = Fault
//
// Machine "state" groups:
//   0 = IDLE, 1 = ENABLE, 2 = WAIT_EN, 3 = RAMP_EN, 4 = RUN, 5 = STOPPING, 10 = FAULT
// Priority rule (for motors): Fault > Running > Starting > Idle
// ──────────────────────────────────────────────────────────────────────────────
VAR CONSTANT
    STATUS_IDLE     : INT := 0;
    STATUS_STARTING : INT := 1;
    STATUS_RUNNING  : INT := 2;
    STATUS_FAULT    : INT := 3;
END_VAR
(*
// ─────────────── Group machine states into a single HMI statusCode ───────────
CASE state OF
    10: // FAULT
        statusCode := STATUS_FAULT;
    4:  // RUN
        statusCode := STATUS_RUNNING;
    1, 2, 3: // ENABLE / WAIT_EN / RAMP_EN
        statusCode := STATUS_STARTING;
ELSE   // IDLE, STOPPING, or any other
        statusCode := STATUS_IDLE;
END_CASE;


// ─────────────── Per-drive status (priority: Fault > Running > Starting > Idle) ───────────────
// FIRST PRESS (MASTER)
IF firstPressVfdFaultFeedback THEN
    firstPressStatusCode := STATUS_FAULT;
ELSIF firstPressVfdRunFeedback THEN
    firstPressStatusCode := STATUS_RUNNING;
ELSIF firstPressDriveEnable THEN
    firstPressStatusCode := STATUS_STARTING;
ELSE
    firstPressStatusCode := STATUS_IDLE;
END_IF;

// SECOND PRESS (SLAVE)
IF secondPressVfdFaultFeedback THEN
    secondPressStatusCode := STATUS_FAULT;
ELSIF secondPressVfdRunFeedback THEN
    secondPressStatusCode := STATUS_RUNNING;
ELSIF secondPressDriveEnable THEN
    secondPressStatusCode := STATUS_STARTING;
ELSE
    secondPressStatusCode := STATUS_IDLE;
END_IF;
*)
END_METHOD

END_FUNCTION_BLOCK

// ---- POUs/Implicit Checks/CheckDivDInt.TcPOU
// Implicitly generated code : DO NOT EDIT
FUNCTION CheckDivDInt : DINT
VAR_INPUT
	divisor:DINT;
END_VAR

// Implicitly generated code : Only an Implementation suggestion
{noflow}
IF divisor = 0 THEN
	CheckDivDInt:=1;
	
	divisionCheckCounter:= divisionCheckCounter + 1;
	
	
ELSE
	CheckDivDInt:=divisor;
END_IF;
{flow}

END_FUNCTION

// ---- POUs/Implicit Checks/CheckDivLInt.TcPOU
// Implicitly generated code : DO NOT EDIT
FUNCTION CheckDivLInt : LINT
VAR_INPUT
	divisor:LINT;
END_VAR

// Implicitly generated code : Only an Implementation suggestion
{noflow}
IF divisor = 0 THEN
	CheckDivLInt:=1;
		divisionCheckCounter:= divisionCheckCounter + 1;

ELSE
	CheckDivLInt:=divisor;
END_IF;
{flow}

END_FUNCTION

// ---- POUs/Implicit Checks/CheckRangeUnsigned.TcPOU
// Implicitly generated code : DO NOT EDIT
FUNCTION CheckRangeUnsigned : UDINT
VAR_INPUT
	value, lower, upper: UDINT;
END_VAR

// Implicitly generated code : Only an Implementation suggestion
{noflow}
IF (value < lower) THEN
	CheckRangeUnsigned := lower;
ELSIF(value > upper) THEN
	CheckRangeUnsigned := upper;
ELSE
	CheckRangeUnsigned := value;
END_IF
{flow}

END_FUNCTION
